REGION Network 6: #Do06 spare2
   RUNG wire#powerrail
      #Do06(Cmd :=, SimulationOn :=, MotorFeedbackInputSelection :=, MotorFeedbackInput :=, WaterSensorSelection :=, WaterSensorInput :=, AlwaysTrue := "AlwaysTRUE", AlwaysFalse := "AlwaysFALSE", OpenClose :=, Spare_3 :=, ValveFeedbackInputSelection :=, ValveFeedbackInput :=, Interlock := #Interlock, FBCheckDelay :=, WSCheckDelay :=, secs := "Sec_Pulse", AlarmAck :=, ModeSel :=, Fault :=, Reset :=, spare :=, spare_1 :=, spare_2 :=, OpFbTrip :=, OpWaterSensorTrip :=, FBCheckActualTime :=, WSCheckActualTime :=, Output =>, FeedBackTripAlarm =>, NoWaterFlowAlarm =>, LineColour =>, ValveColour =>, Mode =>, Status =>)
   END_RUNG
   // the same network as SCL:
   #Do06(AlwaysTrue := "AlwaysTRUE", AlwaysFalse := "AlwaysFALSE", Interlock := #Interlock, secs := "Sec_Pulse");   // "DigitalOutput"
END_REGION

REGION Network 7: #Do07spare3
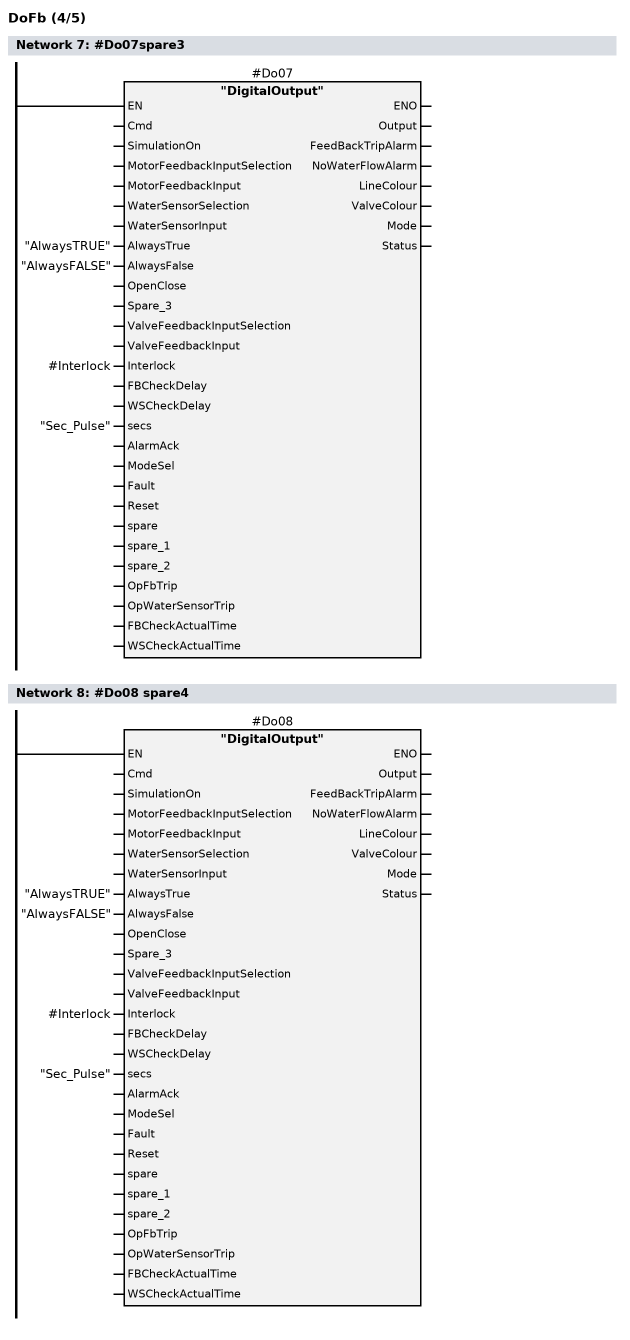
   RUNG wire#powerrail
      #Do07(Cmd :=, SimulationOn :=, MotorFeedbackInputSelection :=, MotorFeedbackInput :=, WaterSensorSelection :=, WaterSensorInput :=, AlwaysTrue := "AlwaysTRUE", AlwaysFalse := "AlwaysFALSE", OpenClose :=, Spare_3 :=, ValveFeedbackInputSelection :=, ValveFeedbackInput :=, Interlock := #Interlock, FBCheckDelay :=, WSCheckDelay :=, secs := "Sec_Pulse", AlarmAck :=, ModeSel :=, Fault :=, Reset :=, spare :=, spare_1 :=, spare_2 :=, OpFbTrip :=, OpWaterSensorTrip :=, FBCheckActualTime :=, WSCheckActualTime :=, Output =>, FeedBackTripAlarm =>, NoWaterFlowAlarm =>, LineColour =>, ValveColour =>, Mode =>, Status =>)
   END_RUNG
   // the same network as SCL:
   #Do07(AlwaysTrue := "AlwaysTRUE", AlwaysFalse := "AlwaysFALSE", Interlock := #Interlock, secs := "Sec_Pulse");   // "DigitalOutput"
END_REGION

REGION Network 8: #Do08 spare4
   RUNG wire#powerrail
      #Do08(Cmd :=, SimulationOn :=, MotorFeedbackInputSelection :=, MotorFeedbackInput :=, WaterSensorSelection :=, WaterSensorInput :=, AlwaysTrue := "AlwaysTRUE", AlwaysFalse := "AlwaysFALSE", OpenClose :=, Spare_3 :=, ValveFeedbackInputSelection :=, ValveFeedbackInput :=, Interlock := #Interlock, FBCheckDelay :=, WSCheckDelay :=, secs := "Sec_Pulse", AlarmAck :=, ModeSel :=, Fault :=, Reset :=, spare :=, spare_1 :=, spare_2 :=, OpFbTrip :=, OpWaterSensorTrip :=, FBCheckActualTime :=, WSCheckActualTime :=, Output =>, FeedBackTripAlarm =>, NoWaterFlowAlarm =>, LineColour =>, ValveColour =>, Mode =>, Status =>)
   END_RUNG
   // the same network as SCL:
   #Do08(AlwaysTrue := "AlwaysTRUE", AlwaysFalse := "AlwaysFALSE", Interlock := #Interlock, secs := "Sec_Pulse");   // "DigitalOutput"
END_REGION

REGION Network 9: ##Do09 spare5
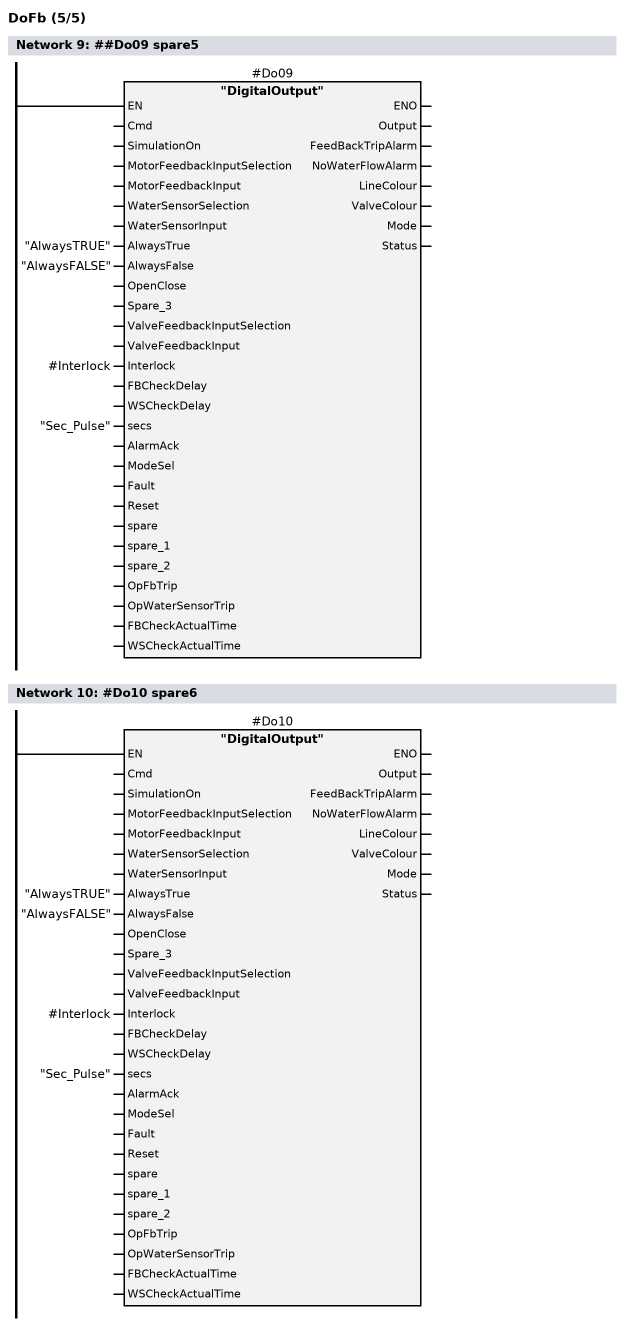
   RUNG wire#powerrail
      #Do09(Cmd :=, SimulationOn :=, MotorFeedbackInputSelection :=, MotorFeedbackInput :=, WaterSensorSelection :=, WaterSensorInput :=, AlwaysTrue := "AlwaysTRUE", AlwaysFalse := "AlwaysFALSE", OpenClose :=, Spare_3 :=, ValveFeedbackInputSelection :=, ValveFeedbackInput :=, Interlock := #Interlock, FBCheckDelay :=, WSCheckDelay :=, secs := "Sec_Pulse", AlarmAck :=, ModeSel :=, Fault :=, Reset :=, spare :=, spare_1 :=, spare_2 :=, OpFbTrip :=, OpWaterSensorTrip :=, FBCheckActualTime :=, WSCheckActualTime :=, Output =>, FeedBackTripAlarm =>, NoWaterFlowAlarm =>, LineColour =>, ValveColour =>, Mode =>, Status =>)
   END_RUNG
   // the same network as SCL:
   #Do09(AlwaysTrue := "AlwaysTRUE", AlwaysFalse := "AlwaysFALSE", Interlock := #Interlock, secs := "Sec_Pulse");   // "DigitalOutput"
END_REGION

REGION Network 10: #Do10 spare6
   RUNG wire#powerrail
      #Do10(Cmd :=, SimulationOn :=, MotorFeedbackInputSelection :=, MotorFeedbackInput :=, WaterSensorSelection :=, WaterSensorInput :=, AlwaysTrue := "AlwaysTRUE", AlwaysFalse := "AlwaysFALSE", OpenClose :=, Spare_3 :=, ValveFeedbackInputSelection :=, ValveFeedbackInput :=, Interlock := #Interlock, FBCheckDelay :=, WSCheckDelay :=, secs := "Sec_Pulse", AlarmAck :=, ModeSel :=, Fault :=, Reset :=, spare :=, spare_1 :=, spare_2 :=, OpFbTrip :=, OpWaterSensorTrip :=, FBCheckActualTime :=, WSCheckActualTime :=, Output =>, FeedBackTripAlarm =>, NoWaterFlowAlarm =>, LineColour =>, ValveColour =>, Mode =>, Status =>)
   END_RUNG
   // the same network as SCL:
   #Do10(AlwaysTrue := "AlwaysTRUE", AlwaysFalse := "AlwaysFALSE", Interlock := #Interlock, secs := "Sec_Pulse");   // "DigitalOutput"
END_REGION
END_FUNCTION_BLOCK

FUNCTION_BLOCK "DigitalOutput"   // FB4, LAD
TITLE = FB4
{ S7_Optimized_Access := 'FALSE' }
// DIGITAL OUTPUT
// stored: AutoNumber false, SetENOAutomatically false
   VAR_INPUT
      Cmd { ExternalVisible := 'False'} : Bool;
      SimulationOn { ExternalVisible := 'False'} : Bool;
      MotorFeedbackInputSelection { ExternalVisible := 'False'} : Bool;
      MotorFeedbackInput { ExternalVisible := 'False'} : Bool;
      WaterSensorSelection { ExternalVisible := 'False'} : Bool;
      WaterSensorInput { ExternalVisible := 'False'} : Bool;
      AlwaysTrue : Bool;
      AlwaysFalse : Bool;
      OpenClose : Bool;   // For Valve Only
      Spare_3 : Bool;   // For Valve Only
      ValveFeedbackInputSelection { ExternalVisible := 'False'} : Bool;
      ValveFeedbackInput { ExternalVisible := 'False'} : Bool;
      Interlock : Bool;
      FBCheckDelay { ExternalVisible := 'False'} : Int;
      WSCheckDelay { ExternalVisible := 'False'} : Int;
      secs { ExternalVisible := 'False'} : Bool;
      AlarmAck { ExternalVisible := 'False'} : Bool;
      ModeSel : Bool;   // 1=Man/ 0=Auto
      Fault : Bool;
      Reset : Bool;
      spare : Bool;
      spare_1 : Bool;
      spare_2 : Bool;
   END_VAR
   VAR_OUTPUT
      Output { ExternalVisible := 'False'} : Bool;
      FeedBackTripAlarm : Bool;
      NoWaterFlowAlarm : Bool;
      LineColour : DInt;
      ValveColour : DInt;
      Mode : DInt;   // Auto=0 , Manual=1
      Status : DInt;
   END_VAR
   VAR_IN_OUT
      OpFbTrip { ExternalVisible := 'False'} : Bool;
      OpWaterSensorTrip { ExternalVisible := 'False'} : Bool;
      FBCheckActualTime { ExternalVisible := 'False'} : Int;
      WSCheckActualTime { ExternalVisible := 'False'} : Int;
   END_VAR
   VAR
      ResetBtn { S7_SetPoint := 'True'} : TON_TIME;
   END_VAR
   VAR_TEMP   // added for the SCL form of the ladder/FBD networks
      _w1 : Bool;
      _w2 : Bool;
   END_VAR
BEGIN

REGION Network 1: #Output
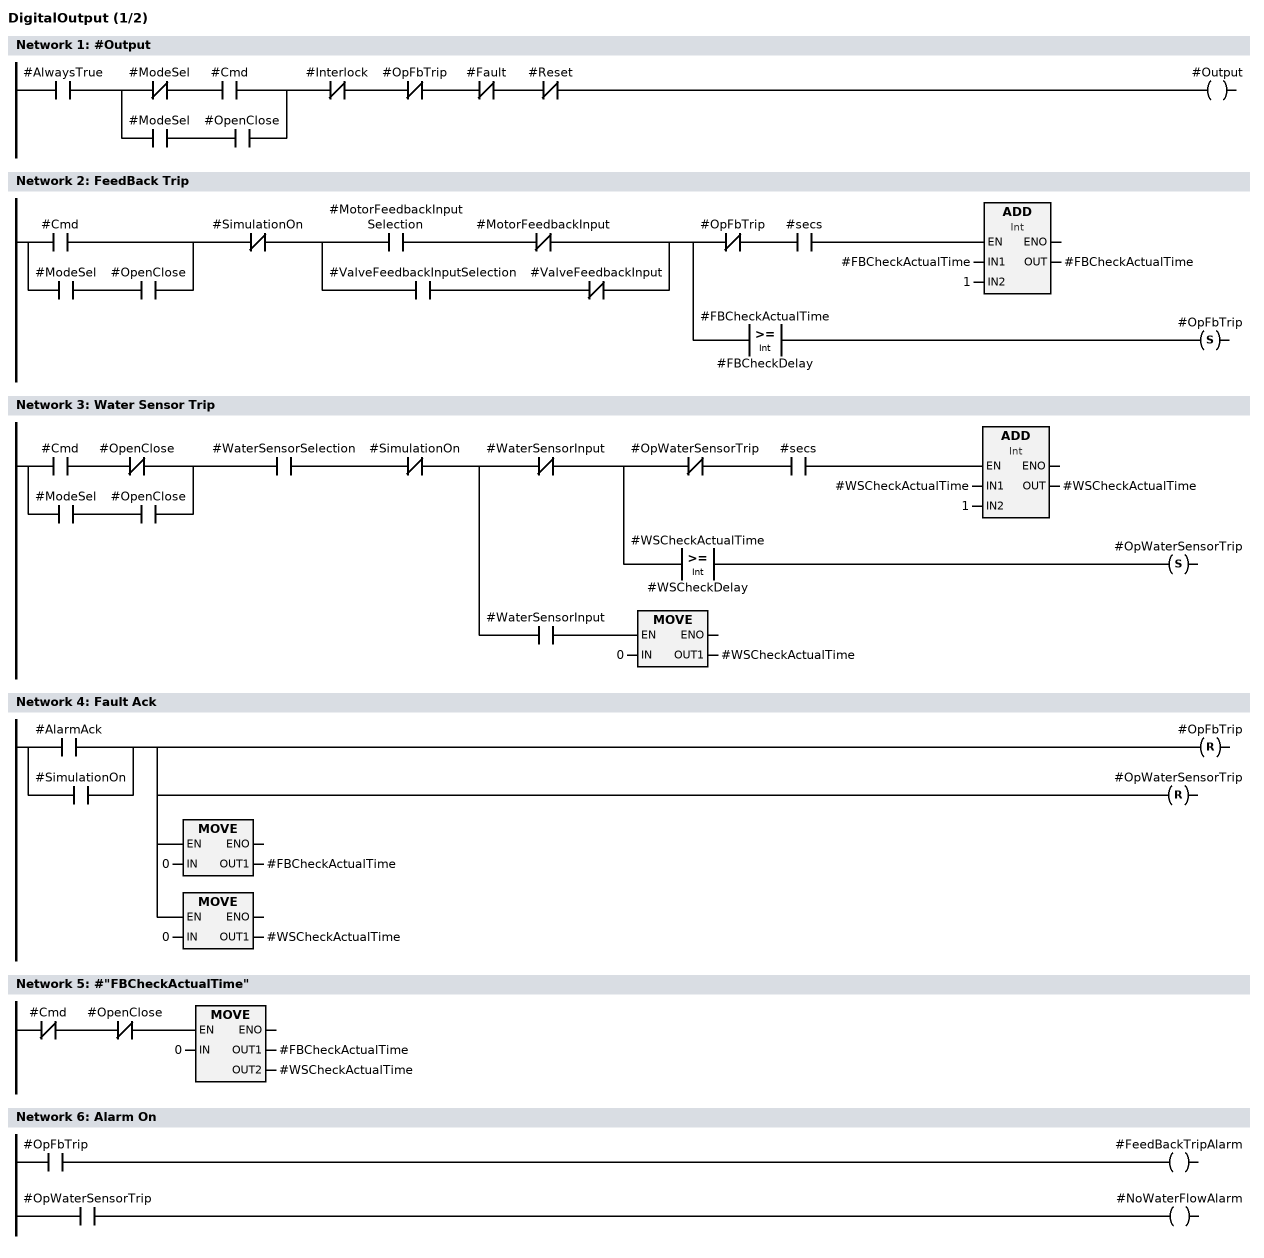
   RUNG wire#powerrail
      Contact( #AlwaysTrue )
      wire#w1
      I_Contact( #ModeSel )
      Contact( #Cmd )
      wire#w2
      I_Contact( #Interlock )
      I_Contact( #OpFbTrip )
      I_Contact( #Fault )
      I_Contact( #Reset )
      Coil( #Output )
   END_RUNG
   RUNG wire#w1
      Contact( #ModeSel )
      Contact( #OpenClose )
   END_RUNG wire#w2
   // the same network as SCL:
   #Output := #AlwaysTrue AND ((NOT #ModeSel AND #Cmd) OR (#ModeSel AND #OpenClose)) AND NOT #Interlock AND NOT #OpFbTrip AND NOT #Fault AND NOT #Reset;
END_REGION

REGION Network 2: FeedBack Trip
   RUNG wire#powerrail
      Contact( #Cmd )
      wire#w1
      I_Contact( #SimulationOn )
      wire#w2
      Contact( #MotorFeedbackInputSelection )
      I_Contact( #MotorFeedbackInput )
      wire#w3
      I_Contact( #OpFbTrip )
      Contact( #secs )
      { S7_Templates := "SrcType := Int"; S7_GenerateENO := "TRUE" } Add(in1 := #FBCheckActualTime, in2 := 1, out => #FBCheckActualTime)
   END_RUNG
   RUNG wire#powerrail
      Contact( #ModeSel )
      Contact( #OpenClose )
   END_RUNG wire#w1
   RUNG wire#w2
      Contact( #ValveFeedbackInputSelection )
      I_Contact( #ValveFeedbackInput )
   END_RUNG wire#w3
   RUNG wire#w3
      { S7_Templates := "SrcType := Int" } GE_Contact(in1 := #FBCheckActualTime, in2 := #FBCheckDelay)
      S_Coil( #OpFbTrip )
   END_RUNG
   // the same network as SCL:
   #_w1 := (#Cmd OR (#ModeSel AND #OpenClose)) AND NOT #SimulationOn AND ((#MotorFeedbackInputSelection AND NOT #MotorFeedbackInput) OR (#ValveFeedbackInputSelection AND NOT #ValveFeedbackInput));
   IF #_w1 AND NOT #OpFbTrip AND #secs THEN #FBCheckActualTime := #FBCheckActualTime + 1; END_IF;
   IF #_w1 AND (#FBCheckActualTime >= #FBCheckDelay) THEN #OpFbTrip := TRUE; END_IF;
END_REGION

REGION Network 3: Water Sensor Trip
   RUNG wire#powerrail
      Contact( #Cmd )
      I_Contact( #OpenClose )
      wire#w1
      Contact( #WaterSensorSelection )
      I_Contact( #SimulationOn )
      wire#w2
      I_Contact( #WaterSensorInput )
      wire#w3
      I_Contact( #OpWaterSensorTrip )
      Contact( #secs )
      { S7_Templates := "SrcType := Int"; S7_GenerateENO := "TRUE" } Add(in1 := #WSCheckActualTime, in2 := 1, out => #WSCheckActualTime)
   END_RUNG
   RUNG wire#powerrail
      Contact( #ModeSel )
      Contact( #OpenClose )
   END_RUNG wire#w1
   RUNG wire#w3
      { S7_Templates := "SrcType := Int" } GE_Contact(in1 := #WSCheckActualTime, in2 := #WSCheckDelay)
      S_Coil( #OpWaterSensorTrip )
   END_RUNG
   RUNG wire#w2
      Contact( #WaterSensorInput )
      { S7_GenerateENO := "TRUE" } Move(in := 0, out1 => #WSCheckActualTime)
   END_RUNG
   // the same network as SCL:
   #_w1 := ((#Cmd AND NOT #OpenClose) OR (#ModeSel AND #OpenClose)) AND #WaterSensorSelection AND NOT #SimulationOn;
   #_w2 := #_w1 AND NOT #WaterSensorInput;
   IF #_w2 AND NOT #OpWaterSensorTrip AND #secs THEN #WSCheckActualTime := #WSCheckActualTime + 1; END_IF;
   IF #_w2 AND (#WSCheckActualTime >= #WSCheckDelay) THEN #OpWaterSensorTrip := TRUE; END_IF;
   IF #_w1 AND #WaterSensorInput THEN #WSCheckActualTime := 0; END_IF;
END_REGION

REGION Network 4: Fault Ack
   RUNG wire#powerrail
      Contact( #AlarmAck )
      wire#w1
      R_Coil( #OpFbTrip )
   END_RUNG
   RUNG wire#powerrail
      Contact( #SimulationOn )
   END_RUNG wire#w1
   RUNG wire#w1
      R_Coil( #OpWaterSensorTrip )
   END_RUNG
   RUNG wire#w1
      { S7_GenerateENO := "TRUE" } Move(in := 0, out1 => #FBCheckActualTime)
   END_RUNG
   RUNG wire#w1
      { S7_GenerateENO := "TRUE" } Move(in := 0, out1 => #WSCheckActualTime)
   END_RUNG
   // the same network as SCL:
   IF #AlarmAck OR #SimulationOn THEN
       #OpFbTrip := FALSE;
       #OpWaterSensorTrip := FALSE;
       #FBCheckActualTime := 0;
       #WSCheckActualTime := 0;
   END_IF;
END_REGION

REGION Network 5: #"FBCheckActualTime"
   RUNG wire#powerrail
      I_Contact( #Cmd )
      I_Contact( #OpenClose )
      { S7_GenerateENO := "TRUE" } Move(in := 0, out1 => #FBCheckActualTime, out2 => #WSCheckActualTime)
   END_RUNG
   // the same network as SCL:
   IF NOT #Cmd AND NOT #OpenClose THEN
       #FBCheckActualTime := 0;
       #WSCheckActualTime := 0;
   END_IF;
END_REGION

REGION Network 6: Alarm On
   RUNG wire#powerrail
      Contact( #OpFbTrip )
      Coil( #FeedBackTripAlarm )
   END_RUNG
   RUNG wire#powerrail
      Contact( #OpWaterSensorTrip )
      Coil( #NoWaterFlowAlarm )
   END_RUNG
   // the same network as SCL:
   #FeedBackTripAlarm := #OpFbTrip;
   #NoWaterFlowAlarm := #OpWaterSensorTrip;
END_REGION

REGION Network 7: Valve Colour
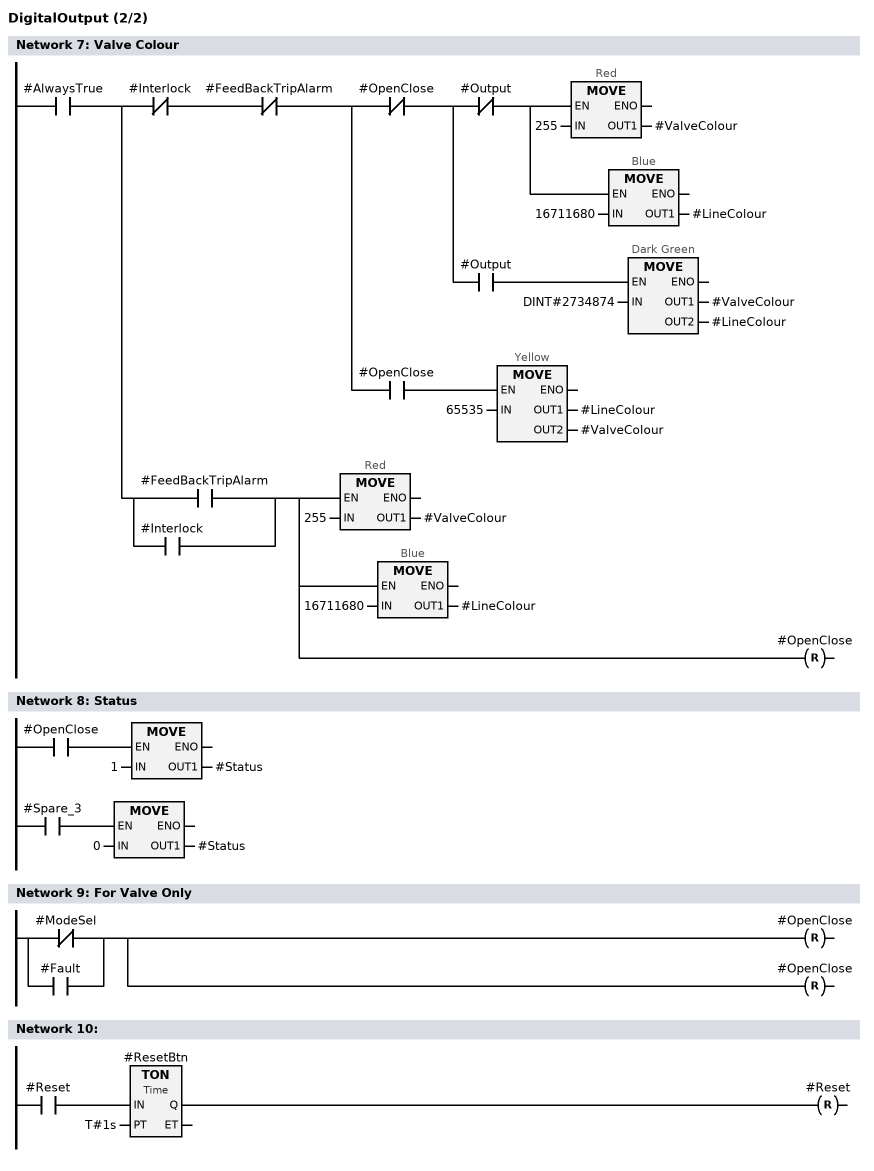
   RUNG wire#powerrail
      Contact( #AlwaysTrue )
      wire#w1
      I_Contact( #Interlock )
      I_Contact( #FeedBackTripAlarm )
      wire#w2
      I_Contact( #OpenClose )
      wire#w3
      I_Contact( #Output )
      wire#w4
      Move(in := 255, out1 => #ValveColour)   // Red
   END_RUNG
   RUNG wire#w4
      Move(in := 16711680, out1 => #LineColour)   // Blue
   END_RUNG
   RUNG wire#w3
      Contact( #Output )
      Move(in := DINT#2734874, out1 => #ValveColour, out2 => #LineColour)   // Dark Green
   END_RUNG
   RUNG wire#w2
      Contact( #OpenClose )
      Move(in := 65535, out1 => #LineColour, out2 => #ValveColour)   // Yellow
   END_RUNG
   RUNG wire#w1
      Contact( #FeedBackTripAlarm )
      wire#w5
      Move(in := 255, out1 => #ValveColour)   // Red
   END_RUNG
   RUNG wire#w1
      Contact( #Interlock )
   END_RUNG wire#w5
   RUNG wire#w5
      Move(in := 16711680, out1 => #LineColour)   // Blue
   END_RUNG
   RUNG wire#w5
      R_Coil( #OpenClose )
   END_RUNG
   // the same network as SCL:
   #_w1 := #AlwaysTrue AND NOT #Interlock AND NOT #FeedBackTripAlarm;
   #_w2 := #_w1 AND NOT #OpenClose;
   IF #_w2 AND NOT #Output THEN
       #ValveColour := 255;   // Red
       #LineColour := 16711680;   // Blue
   END_IF;
   IF #_w2 AND #Output THEN
       #ValveColour := DINT#2734874;   // Dark Green
       #LineColour := DINT#2734874;
   END_IF;
   IF #_w1 AND #OpenClose THEN
       #LineColour := 65535;   // Yellow
       #ValveColour := 65535;
   END_IF;
   IF #AlwaysTrue AND (#FeedBackTripAlarm OR #Interlock) THEN
       #ValveColour := 255;   // Red
       #LineColour := 16711680;   // Blue
       #OpenClose := FALSE;
   END_IF;
END_REGION

REGION Network 8: Status
   RUNG wire#powerrail
      Contact( #OpenClose )
      Move(in := 1, out1 => #Status)
   END_RUNG
   RUNG wire#powerrail
      Contact( #Spare_3 )
      Move(in := 0, out1 => #Status)
   END_RUNG
   // the same network as SCL:
   IF #OpenClose THEN #Status := 1; END_IF;
   IF #Spare_3 THEN #Status := 0; END_IF;
END_REGION

REGION Network 9: For Valve Only
   RUNG wire#powerrail
      I_Contact( #ModeSel )
      wire#w1
      R_Coil( #OpenClose )
   END_RUNG
   RUNG wire#powerrail
      Contact( #Fault )
   END_RUNG wire#w1
   RUNG wire#w1
      R_Coil( #OpenClose )
   END_RUNG
   // the same network as SCL:
   IF NOT #ModeSel OR #Fault THEN
       #OpenClose := FALSE;
       #OpenClose := FALSE;
   END_IF;
END_REGION

REGION Network 10
   RUNG wire#powerrail
      Contact( #Reset )
      { S7_Templates := "time_type := Time" } #ResetBtn.TON(pt := T#1s, et =>)
      R_Coil( #Reset )
   END_RUNG
   // the same network as SCL:
   #ResetBtn(IN := #Reset, PT := T#1s);   // TON
   IF #ResetBtn.Q THEN #Reset := FALSE; END_IF;
END_REGION
END_FUNCTION_BLOCK

FUNCTION_BLOCK "TIMER"   // FB6, LAD
{ S7_Optimized_Access := 'FALSE' }
// stored: SetENOAutomatically false
   VAR_INPUT
      TIME_START : Bool;
      TIME_PULSE : Bool;
      TIME_TRSET : Bool;
      MINI_ENABLE : Bool;
      TIME_IN_MINI : DInt;
      TIME_IN_SEC : DInt;
   END_VAR
   VAR_OUTPUT
      DONE_BIT : Bool;
      ES_MINIT : DInt;
      ES_SEC : DInt;
   END_VAR
   VAR_IN_OUT
      TEMP_1 : DInt;
      TEMP_5 : DInt;
      TEMP_2 : DInt;
      TEMP_3 : DInt;
      TEMP_BIT_1 : Bool;
      TEMP_BIT_2 : Bool;
   END_VAR
   VAR_TEMP   // added for the SCL form of the ladder/FBD networks
      _w1 : Bool;
   END_VAR
BEGIN

REGION Network 1
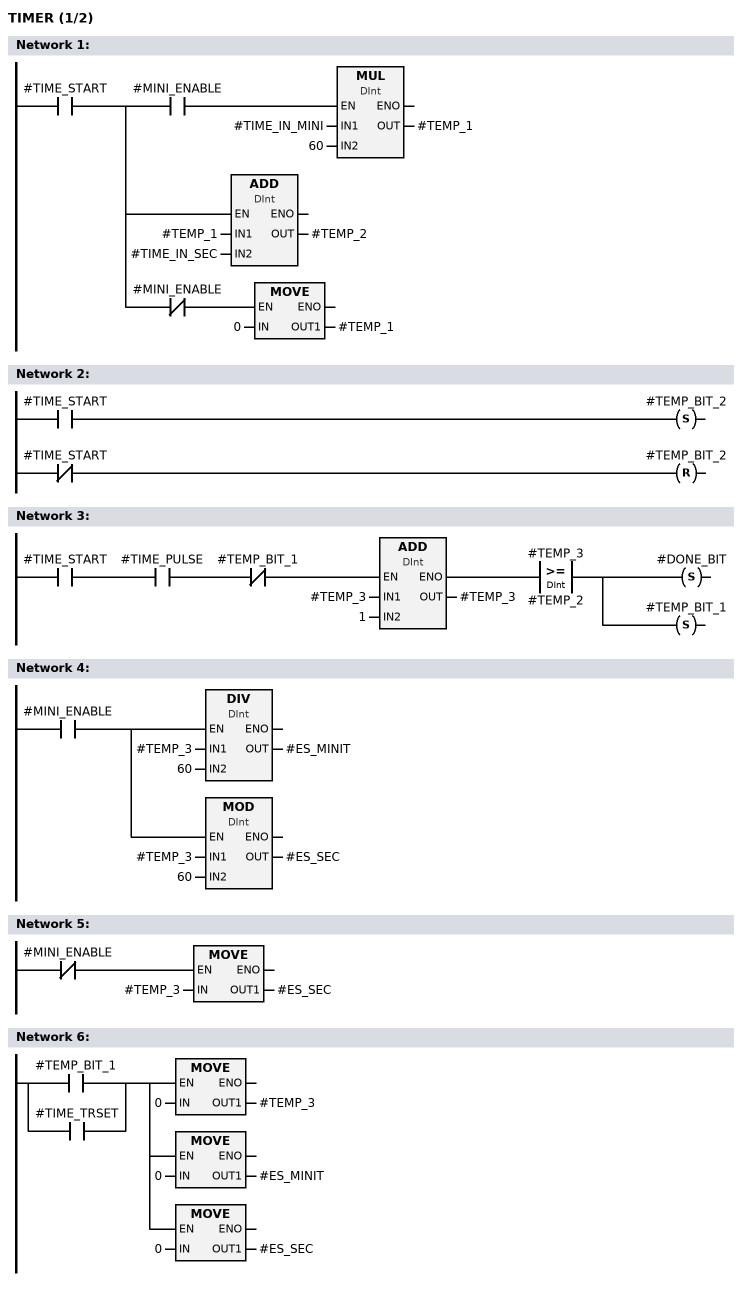
   RUNG wire#powerrail
      Contact( #TIME_START )
      wire#w1
      Contact( #MINI_ENABLE )
      { S7_Templates := "SrcType := DInt"; S7_GenerateENO := "TRUE" } Mul(in1 := #TIME_IN_MINI, in2 := 60, out => #TEMP_1)
   END_RUNG
   RUNG wire#w1
      { S7_Templates := "SrcType := DInt"; S7_GenerateENO := "TRUE" } Add(in1 := #TEMP_1, in2 := #TIME_IN_SEC, out => #TEMP_2)
   END_RUNG
   RUNG wire#w1
      I_Contact( #MINI_ENABLE )
      { S7_GenerateENO := "TRUE" } Move(in := 0, out1 => #TEMP_1)
   END_RUNG
   // the same network as SCL:
   IF #TIME_START AND #MINI_ENABLE THEN #TEMP_1 := #TIME_IN_MINI * 60; END_IF;
   IF #TIME_START THEN #TEMP_2 := #TEMP_1 + #TIME_IN_SEC; END_IF;
   IF #TIME_START AND NOT #MINI_ENABLE THEN #TEMP_1 := 0; END_IF;
END_REGION

REGION Network 2
   RUNG wire#powerrail
      Contact( #TIME_START )
      S_Coil( #TEMP_BIT_2 )
   END_RUNG
   RUNG wire#powerrail
      I_Contact( #TIME_START )
      R_Coil( #TEMP_BIT_2 )
   END_RUNG
   // the same network as SCL:
   IF #TIME_START THEN #TEMP_BIT_2 := TRUE; END_IF;
   IF NOT #TIME_START THEN #TEMP_BIT_2 := FALSE; END_IF;
END_REGION

REGION Network 3
   RUNG wire#powerrail
      Contact( #TIME_START )
      Contact( #TIME_PULSE )
      I_Contact( #TEMP_BIT_1 )
      { S7_Templates := "SrcType := DInt"; S7_GenerateENO := "TRUE" } Add(in1 := #TEMP_3, in2 := 1, out => #TEMP_3)
      { S7_Templates := "SrcType := DInt" } GE_Contact(in1 := #TEMP_3, in2 := #TEMP_2)
      wire#w1
      S_Coil( #DONE_BIT )
   END_RUNG
   RUNG wire#w1
      S_Coil( #TEMP_BIT_1 )
   END_RUNG
   // the same network as SCL:
   // ENO of a box is taken as its EN; it also drops when the box reports an error
   #_w1 := #TIME_START AND #TIME_PULSE AND NOT #TEMP_BIT_1;
   IF #_w1 THEN #TEMP_3 := #TEMP_3 + 1; END_IF;
   IF #_w1 AND (#TEMP_3 >= #TEMP_2) THEN
       #DONE_BIT := TRUE;
       #TEMP_BIT_1 := TRUE;
   END_IF;
END_REGION

REGION Network 4
   RUNG wire#powerrail
      Contact( #MINI_ENABLE )
      wire#w1
      { S7_Templates := "SrcType := DInt"; S7_GenerateENO := "TRUE" } Div(in1 := #TEMP_3, in2 := 60, out => #ES_MINIT)
   END_RUNG
   RUNG wire#w1
      { S7_Templates := "SrcType := DInt"; S7_GenerateENO := "TRUE" } Mod(in1 := #TEMP_3, in2 := 60, out => #ES_SEC)
   END_RUNG
   // the same network as SCL:
   IF #MINI_ENABLE THEN
       #ES_MINIT := #TEMP_3 / 60;
       #ES_SEC := #TEMP_3 MOD 60;
   END_IF;
END_REGION

REGION Network 5
   RUNG wire#powerrail
      I_Contact( #MINI_ENABLE )
      { S7_GenerateENO := "TRUE" } Move(in := #TEMP_3, out1 => #ES_SEC)
   END_RUNG
   // the same network as SCL:
   IF NOT #MINI_ENABLE THEN #ES_SEC := #TEMP_3; END_IF;
END_REGION

REGION Network 6
   RUNG wire#powerrail
      Contact( #TEMP_BIT_1 )
      wire#w1
      { S7_GenerateENO := "TRUE" } Move(in := 0, out1 => #TEMP_3)
   END_RUNG
   RUNG wire#powerrail
      Contact( #TIME_TRSET )
   END_RUNG wire#w1
   RUNG wire#w1
      { S7_GenerateENO := "TRUE" } Move(in := 0, out1 => #ES_MINIT)
   END_RUNG
   RUNG wire#w1
      { S7_GenerateENO := "TRUE" } Move(in := 0, out1 => #ES_SEC)
   END_RUNG
   // the same network as SCL:
   IF #TEMP_BIT_1 OR #TIME_TRSET THEN
       #TEMP_3 := 0;
       #ES_MINIT := 0;
       #ES_SEC := 0;
   END_IF;
END_REGION

REGION Network 7
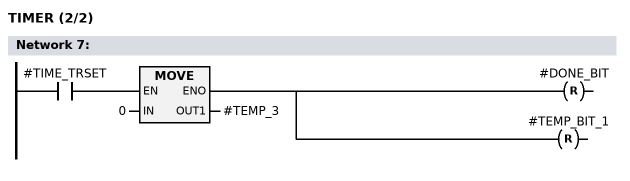
   RUNG wire#powerrail
      Contact( #TIME_TRSET )
      { S7_GenerateENO := "TRUE" } Move(in := 0, out1 => #TEMP_3)
      wire#w1
      R_Coil( #DONE_BIT )
   END_RUNG
   RUNG wire#w1
      R_Coil( #TEMP_BIT_1 )
   END_RUNG
   // the same network as SCL:
   // ENO of a box is taken as its EN; it also drops when the box reports an error
   IF #TIME_TRSET THEN
       #TEMP_3 := 0;
       #DONE_BIT := FALSE;
       #TEMP_BIT_1 := FALSE;
   END_IF;
END_REGION
END_FUNCTION_BLOCK

FUNCTION "FaceplateFc" : Void   // FC102, LAD
{ S7_Optimized_Access := 'TRUE' }
// stored: AutoNumber false, SetENOAutomatically false
BEGIN

REGION Network 1 (SCL): Valve Open
   "ValveManualMode".Cv01 := "DO_FaceplateDb".Cv01.ValveOpen;
   "ValveManualMode".Cv01 := "DO_FaceplateDb".Cv01.ValveOpen;
   "ValveManualMode".Cv02 := "DO_FaceplateDb".Cv02.ValveOpen;
   "ValveManualMode".Cv03 := "DO_FaceplateDb".Cv03.ValveOpen;
   "ValveManualMode".Cv04 := "DO_FaceplateDb".Cv04.ValveOpen;
   "ValveManualMode".Cv05 := "DO_FaceplateDb".Cv05.ValveOpen;
   "ValveManualMode".Cv06 := "DO_FaceplateDb".Cv06.ValveOpen;
   "ValveManualMode".Cv07 := "DO_FaceplateDb".Cv07.ValveOpen;
   "ValveManualMode".Cv08 := "DO_FaceplateDb".Cv08.ValveOpen;
   "ValveManualMode".Cv09 := "DO_FaceplateDb".Cv09.ValveOpen;
   "ValveManualMode".Cv10 := "DO_FaceplateDb".Cv10.ValveOpen;
   "ValveManualMode".Cv11 := "DO_FaceplateDb".Cv11.ValveOpen;
   "ValveManualMode".Cv12 := "DO_FaceplateDb".Cv12.ValveOpen;
   "ValveManualMode".Cv13 := "DO_FaceplateDb".Cv13.ValveOpen;
   "ValveManualMode".Cv14 := "DO_FaceplateDb".Cv14.ValveOpen;
   "ValveManualMode".Cv15 := "DO_FaceplateDb".Cv15.ValveOpen;
   "ValveManualMode".Cv16 := "DO_FaceplateDb".Cv16.ValveOpen;
   "ValveManualMode".Cv17 := "DO_FaceplateDb".Cv17.ValveOpen;
   "ValveManualMode".Cv18 := "DO_FaceplateDb".Cv18.ValveOpen;
   "ValveManualMode".Cv19 := "DO_FaceplateDb".Cv19.ValveOpen;
   "ValveManualMode".Cv20 := "DO_FaceplateDb".Cv20.ValveOpen;
   "ValveManualMode".Cv21 := "DO_FaceplateDb".Cv21.ValveOpen;
   "ValveManualMode".Cv22 := "DO_FaceplateDb".Cv22.ValveOpen;
   "ValveManualMode".Cv23 := "DO_FaceplateDb".Cv23.ValveOpen;
   "ValveManualMode".Cv24 := "DO_FaceplateDb".Cv24.ValveOpen;
   "ValveManualMode".Cv25 := "DO_FaceplateDb".Cv25.ValveOpen;
   "ValveManualMode".Cv26 := "DO_FaceplateDb".Cv26.ValveOpen;
   "ValveManualMode".Cv27 := "DO_FaceplateDb".Cv27.ValveOpen;
   "ValveManualMode".Cv28 := "DO_FaceplateDb".Cv28.ValveOpen;
   "ValveManualMode".Cv29 := "DO_FaceplateDb".Cv29.ValveOpen;
   "ValveManualMode".Cv30 := "DO_FaceplateDb".Cv30.ValveOpen;
   "ValveManualMode".Cv31 := "DO_FaceplateDb".Cv31.ValveOpen;
   "ValveManualMode".Cv32 := "DO_FaceplateDb".Cv32.ValveOpen;
   "ValveManualMode".Cv33 := "DO_FaceplateDb".Cv33.ValveOpen;
   "ValveManualMode".Cv34 := "DO_FaceplateDb".Cv34.ValveOpen;
   "ValveManualMode".Cv35 := "DO_FaceplateDb".Cv35.ValveOpen;
   "ValveManualMode".Cv36 := "DO_FaceplateDb".Cv36.ValveOpen;
   "ValveManualMode".Cv37 := "DO_FaceplateDb".Cv37.ValveOpen;
   "ValveManualMode".Cv38 := "DO_FaceplateDb".Cv38.ValveOpen;
   "ValveManualMode".Cv39 := "DO_FaceplateDb".Cv39.ValveOpen;
   "ValveManualMode".Cv40 := "DO_FaceplateDb".Cv40.ValveOpen;
   "ValveManualMode".Cv41 := "DO_FaceplateDb".Cv41.ValveOpen;
   "ValveManualMode".Cv42 := "DO_FaceplateDb".Cv42.ValveOpen;
   "ValveManualMode".Cv43 := "DO_FaceplateDb".Cv43.ValveOpen;
   "ValveManualMode".Cv44 := "DO_FaceplateDb".Cv44.ValveOpen;
   "ValveManualMode".Cv45 := "DO_FaceplateDb".Cv45.ValveOpen;
   "ValveManualMode".Cv46 := "DO_FaceplateDb".Cv46.ValveOpen;
   "ValveManualMode".Cv47 := "DO_FaceplateDb".Cv47.ValveOpen;
   "ValveManualMode".Cv48 := "DO_FaceplateDb".Cv48.ValveOpen;
   "ValveManualMode".Cv49 := "DO_FaceplateDb".Cv49.ValveOpen;
   "ValveManualMode".Cv50 := "DO_FaceplateDb".Cv50.ValveOpen;
   "ValveManualMode".Cv51 := "DO_FaceplateDb".Cv51.ValveOpen;
   "ValveManualMode".Cv52 := "DO_FaceplateDb".Cv52.ValveOpen;
   "ValveManualMode".Cv53 := "DO_FaceplateDb".Cv53.ValveOpen;
   "ValveManualMode".Cv54 := "DO_FaceplateDb".Cv54.ValveOpen;
   "ValveManualMode".Cv55 := "DO_FaceplateDb".Cv55.ValveOpen;
   "ValveManualMode".Cv56 := "DO_FaceplateDb".Cv56.ValveOpen;
   "ValveManualMode".Cv57 := "DO_FaceplateDb".Cv57.ValveOpen;
   "ValveManualMode".Cv58 := "DO_FaceplateDb".Cv58.ValveOpen;
   "ValveManualMode".Cv59 := "DO_FaceplateDb".Cv59.ValveOpen;
   "ValveManualMode".Cv60 := "DO_FaceplateDb".Cv60.ValveOpen;
   "ValveManualMode".Cv61 := "DO_FaceplateDb".Cv61.ValveOpen;
   "ValveManualMode".Cv62 := "DO_FaceplateDb".Cv62.ValveOpen;
   "ValveManualMode".Cv63 := "DO_FaceplateDb".Cv63.ValveOpen;
   "ValveManualMode".Cv64 := "DO_FaceplateDb".Cv64.ValveOpen;
   "ValveManualMode".Fbov01 := "DO_FaceplateDb".Fbov01.ValveOpen;
END_REGION

REGION Network 2 (SCL): Pump Command
   "DoManualModeDb".Mm01Cmd :="DO_FaceplateDb"."Mm01 Ref".ValveOpen;
   "DoManualModeDb".Cp01Cmd := "DO_FaceplateDb"."Cp01 Ref".ValveOpen;


   //"DoDb".Do01.OpenClose := "DO_FaceplateDb"."Mm01 Ref".ValveOpen;
   //"DoDb".Do02.OpenClose := "DO_FaceplateDb"."Cp01 Ref".ValveOpen;
END_REGION

REGION Network 3 (SCL): Analog Output
   //Actual Rpm

   "Ao_Faceplate_Db".Mm01Ref.ActualRpm := "AoDb".Ao01.ActualRpm;
   "Ao_Faceplate_Db".Cp01Ref.ActualRpm:= "AoDb".Ao02.ActualRpm;


   //Min. Opeating Rpm
   // "AoDb".Ao01.MinOperatingRpm := "Ao_Faceplate_Db".CP01.MinOperating;
   //"AoDb".Ao02.MinOperatingRpm := "Ao_Faceplate_Db".MM01.MinOperating;
   "Ao_Faceplate_Db".Mm01Ref.MinOperating:= "AoDb".Ao01.MinOperatingRpm;
   "Ao_Faceplate_Db".Cp01Ref.MinOperating := "AoDb".Ao02.MinOperatingRpm;

   //Max. Operating Rpm
   "Ao_Faceplate_Db".Mm01Ref.MaxOperating:=  "AoDb".Ao01.MaxOperatingRpm;
   "Ao_Faceplate_Db".Cp01Ref.MaxOperating:= "AoDb".Ao02.MaxOperatingRpm;

   //Maximum Rpm
   // "AoDb".Ao01.MaxRpm := "Ao_Faceplate_Db".CP01.Maximum;
   // "AoDb".Ao02.MaxRpm := "Ao_Faceplate_Db".MM01.Maximum;
   "Ao_Faceplate_Db".Mm01Ref.Maximum:= "AoDb".Ao01.MaxRpm;
   "Ao_Faceplate_Db".Cp01Ref.Maximum:= "AoDb".Ao02.MaxRpm;

   //Manual Rpm
   // "AoDb".Ao01.ManualRpm := "Ao_Faceplate_Db".CP01.Manual;
   // "AoDb".Ao02.ManualRpm := "Ao_Faceplate_Db".MM01.Manual;
   "Ao_Faceplate_Db".Mm01Ref.Manual := "AoDb".Ao01.ManualRpm;
   "Ao_Faceplate_Db".Cp01Ref.Manual:= "AoDb".Ao02.ManualRpm;
END_REGION

REGION Network 4 (SCL): Analog Input
   // Moving Int value for units, 0 - Degree Celcius, 1 - bar, 2 - 

   // //"Ai_Faceplate_Db".Ai01.Unit := 0; spare
   // //"Ai_Faceplate_Db".Ai02.Unit := 0; spare
   // "Ai_Faceplate_Db".Ai03.Unit := 0;
   // "Ai_Faceplate_Db".Ai04.Unit := 0;
   // "Ai_Faceplate_Db".Ai05.Unit := 0;
   // "Ai_Faceplate_Db".Ai06.Unit := 0;
   // "Ai_Faceplate_Db".Ai07.Unit := 0;
   // "Ai_Faceplate_Db".Ai08.Unit := 1;
   // "Ai_Faceplate_Db".Ai09.Unit := 2;
   // "Ai_Faceplate_Db".Ai10.Unit := 3;
   // "Ai_Faceplate_Db".Ai11.Unit := 4;
END_REGION

REGION Network 5 (SCL)
   // "ValveDb".Cv01.OpenClose := "DO_FaceplateDb".Cv01.ValveOpen;
END_REGION
END_FUNCTION

FUNCTION "AlarmsFc" : Void   // FC181, LAD
{ S7_Optimized_Access := 'TRUE' }
// stored: AutoNumber false, SetENOAutomatically false
   VAR_TEMP   // added for the SCL form of the ladder/FBD networks
      _w1 : Bool;
      _w2 : Bool;
      _w3 : Bool;
      _w4 : Bool;
      _w5 : Bool;
      _w6 : Bool;
      _w7 : Bool;
      _w8 : Bool;
      _w9 : Bool;
      _w10 : Bool;
      _w11 : Bool;
      _w12 : Bool;
      _w13 : Bool;
      _w14 : Bool;
      _w15 : Bool;
      _w16 : Bool;
      _w17 : Bool;
      _w18 : Bool;
      _w19 : Bool;
      _w20 : Bool;
      _w21 : Bool;
      _w22 : Bool;
      _w23 : Bool;
      _w24 : Bool;
      _w25 : Bool;
      _w26 : Bool;
      _w27 : Bool;
      _w28 : Bool;
      _w29 : Bool;
      _w30 : Bool;
      _w31 : Bool;
      _w32 : Bool;
      _w33 : Bool;
      _w34 : Bool;
      _w35 : Bool;
      _w36 : Bool;
      _w37 : Bool;
      _w38 : Bool;
      _w39 : Bool;
      _w40 : Bool;
      _w41 : Bool;
      _w42 : Bool;
      _w43 : Bool;
      _w44 : Bool;
      _w45 : Bool;
      _w46 : Bool;
   END_VAR
BEGIN

REGION Network 1: "SafetyAlarms".ControlKeyOff
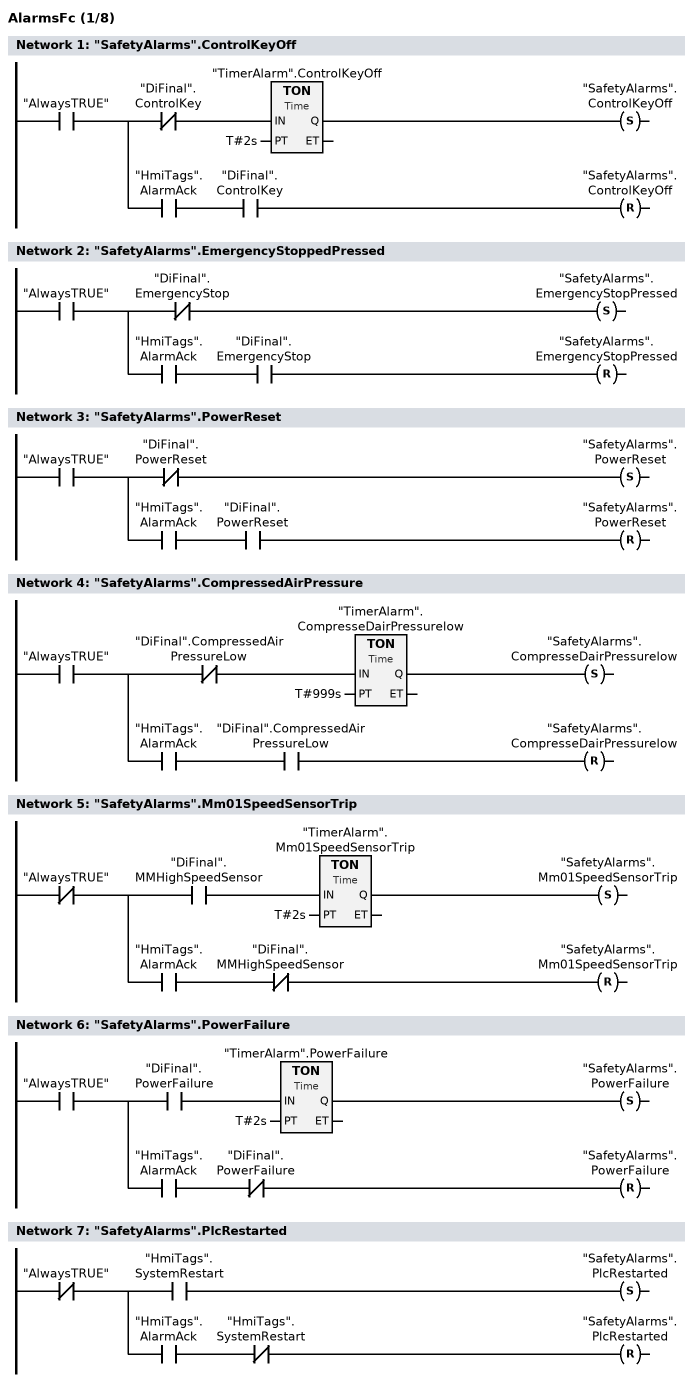
   RUNG wire#powerrail
      Contact( "AlwaysTRUE" )
      wire#w1
      I_Contact( "DiFinal".ControlKey )
      { S7_Templates := "time_type := Time" } "TimerAlarm".ControlKeyOff.TON(pt := T#2s, et =>)
      S_Coil( "SafetyAlarms".ControlKeyOff )
   END_RUNG
   RUNG wire#w1
      Contact( "HmiTags".AlarmAck )
      Contact( "DiFinal".ControlKey )
      R_Coil( "SafetyAlarms".ControlKeyOff )
   END_RUNG
   // the same network as SCL:
   "TimerAlarm".ControlKeyOff.TON(IN := "AlwaysTRUE" AND NOT "DiFinal".ControlKey, PT := T#2s);
   IF "TimerAlarm".ControlKeyOff.Q THEN "SafetyAlarms".ControlKeyOff := TRUE; END_IF;
   IF "AlwaysTRUE" AND "HmiTags".AlarmAck AND "DiFinal".ControlKey THEN
       "SafetyAlarms".ControlKeyOff := FALSE;
   END_IF;
END_REGION

REGION Network 2: "SafetyAlarms".EmergencyStoppedPressed
   RUNG wire#powerrail
      Contact( "AlwaysTRUE" )
      wire#w1
      I_Contact( "DiFinal".EmergencyStop )
      S_Coil( "SafetyAlarms".EmergencyStopPressed )
   END_RUNG
   RUNG wire#w1
      Contact( "HmiTags".AlarmAck )
      Contact( "DiFinal".EmergencyStop )
      R_Coil( "SafetyAlarms".EmergencyStopPressed )
   END_RUNG
   // the same network as SCL:
   IF "AlwaysTRUE" AND NOT "DiFinal".EmergencyStop THEN "SafetyAlarms".EmergencyStopPressed := TRUE; END_IF;
   IF "AlwaysTRUE" AND "HmiTags".AlarmAck AND "DiFinal".EmergencyStop THEN
       "SafetyAlarms".EmergencyStopPressed := FALSE;
   END_IF;
END_REGION

REGION Network 3: "SafetyAlarms".PowerReset
   RUNG wire#powerrail
      Contact( "AlwaysTRUE" )
      wire#w1
      I_Contact( "DiFinal".PowerReset )
      S_Coil( "SafetyAlarms".PowerReset )
   END_RUNG
   RUNG wire#w1
      Contact( "HmiTags".AlarmAck )
      Contact( "DiFinal".PowerReset )
      R_Coil( "SafetyAlarms".PowerReset )
   END_RUNG
   // the same network as SCL:
   IF "AlwaysTRUE" AND NOT "DiFinal".PowerReset THEN "SafetyAlarms".PowerReset := TRUE; END_IF;
   IF "AlwaysTRUE" AND "HmiTags".AlarmAck AND "DiFinal".PowerReset THEN
       "SafetyAlarms".PowerReset := FALSE;
   END_IF;
END_REGION

REGION Network 4: "SafetyAlarms".CompressedAirPressure
   RUNG wire#powerrail
      Contact( "AlwaysTRUE" )
      wire#w1
      I_Contact( "DiFinal".CompressedAirPressureLow )
      { S7_Templates := "time_type := Time" } "TimerAlarm".CompresseDairPressurelow.TON(pt := T#999s, et =>)
      S_Coil( "SafetyAlarms".CompresseDairPressurelow )
   END_RUNG
   RUNG wire#w1
      Contact( "HmiTags".AlarmAck )
      Contact( "DiFinal".CompressedAirPressureLow )
      R_Coil( "SafetyAlarms".CompresseDairPressurelow )
   END_RUNG
   // the same network as SCL:
   "TimerAlarm".CompresseDairPressurelow.TON(IN := "AlwaysTRUE" AND NOT "DiFinal".CompressedAirPressureLow,
                           PT := T#999s);
   IF "TimerAlarm".CompresseDairPressurelow.Q THEN "SafetyAlarms".CompresseDairPressurelow := TRUE; END_IF;
   IF "AlwaysTRUE" AND "HmiTags".AlarmAck AND "DiFinal".CompressedAirPressureLow THEN
       "SafetyAlarms".CompresseDairPressurelow := FALSE;
   END_IF;
END_REGION

REGION Network 5: "SafetyAlarms".Mm01SpeedSensorTrip
   RUNG wire#powerrail
      I_Contact( "AlwaysTRUE" )
      wire#w1
      Contact( "DiFinal".MMHighSpeedSensor )
      { S7_Templates := "time_type := Time" } "TimerAlarm".Mm01SpeedSensorTrip.TON(pt := T#2s, et =>)
      S_Coil( "SafetyAlarms".Mm01SpeedSensorTrip )
   END_RUNG
   RUNG wire#w1
      Contact( "HmiTags".AlarmAck )
      I_Contact( "DiFinal".MMHighSpeedSensor )
      R_Coil( "SafetyAlarms".Mm01SpeedSensorTrip )
   END_RUNG
   // the same network as SCL:
   "TimerAlarm".Mm01SpeedSensorTrip.TON(IN := NOT "AlwaysTRUE" AND "DiFinal".MMHighSpeedSensor, PT := T#2s);
   IF "TimerAlarm".Mm01SpeedSensorTrip.Q THEN "SafetyAlarms".Mm01SpeedSensorTrip := TRUE; END_IF;
   IF NOT "AlwaysTRUE" AND "HmiTags".AlarmAck AND NOT "DiFinal".MMHighSpeedSensor THEN
       "SafetyAlarms".Mm01SpeedSensorTrip := FALSE;
   END_IF;
END_REGION

REGION Network 6: "SafetyAlarms".PowerFailure
   RUNG wire#powerrail
      Contact( "AlwaysTRUE" )
      wire#w1
      Contact( "DiFinal".PowerFailure )
      { S7_Templates := "time_type := Time" } "TimerAlarm".PowerFailure.TON(pt := T#2s, et =>)
      S_Coil( "SafetyAlarms".PowerFailure )
   END_RUNG
   RUNG wire#w1
      Contact( "HmiTags".AlarmAck )
      I_Contact( "DiFinal".PowerFailure )
      R_Coil( "SafetyAlarms".PowerFailure )
   END_RUNG
   // the same network as SCL:
   "TimerAlarm".PowerFailure.TON(IN := "AlwaysTRUE" AND "DiFinal".PowerFailure, PT := T#2s);
   IF "TimerAlarm".PowerFailure.Q THEN "SafetyAlarms".PowerFailure := TRUE; END_IF;
   IF "AlwaysTRUE" AND "HmiTags".AlarmAck AND NOT "DiFinal".PowerFailure THEN
       "SafetyAlarms".PowerFailure := FALSE;
   END_IF;
END_REGION

REGION Network 7: "SafetyAlarms".PlcRestarted
   RUNG wire#powerrail
      I_Contact( "AlwaysTRUE" )
      wire#w1
      Contact( "HmiTags".SystemRestart )
      S_Coil( "SafetyAlarms".PlcRestarted )
   END_RUNG
   RUNG wire#w1
      Contact( "HmiTags".AlarmAck )
      I_Contact( "HmiTags".SystemRestart )
      R_Coil( "SafetyAlarms".PlcRestarted )
   END_RUNG
   // the same network as SCL:
   IF NOT "AlwaysTRUE" AND "HmiTags".SystemRestart THEN "SafetyAlarms".PlcRestarted := TRUE; END_IF;
   IF NOT "AlwaysTRUE" AND "HmiTags".AlarmAck AND NOT "HmiTags".SystemRestart THEN
       "SafetyAlarms".PlcRestarted := FALSE;
   END_IF;
END_REGION

REGION Network 8: "SafetyAlarms".Mm01OverloadTrip
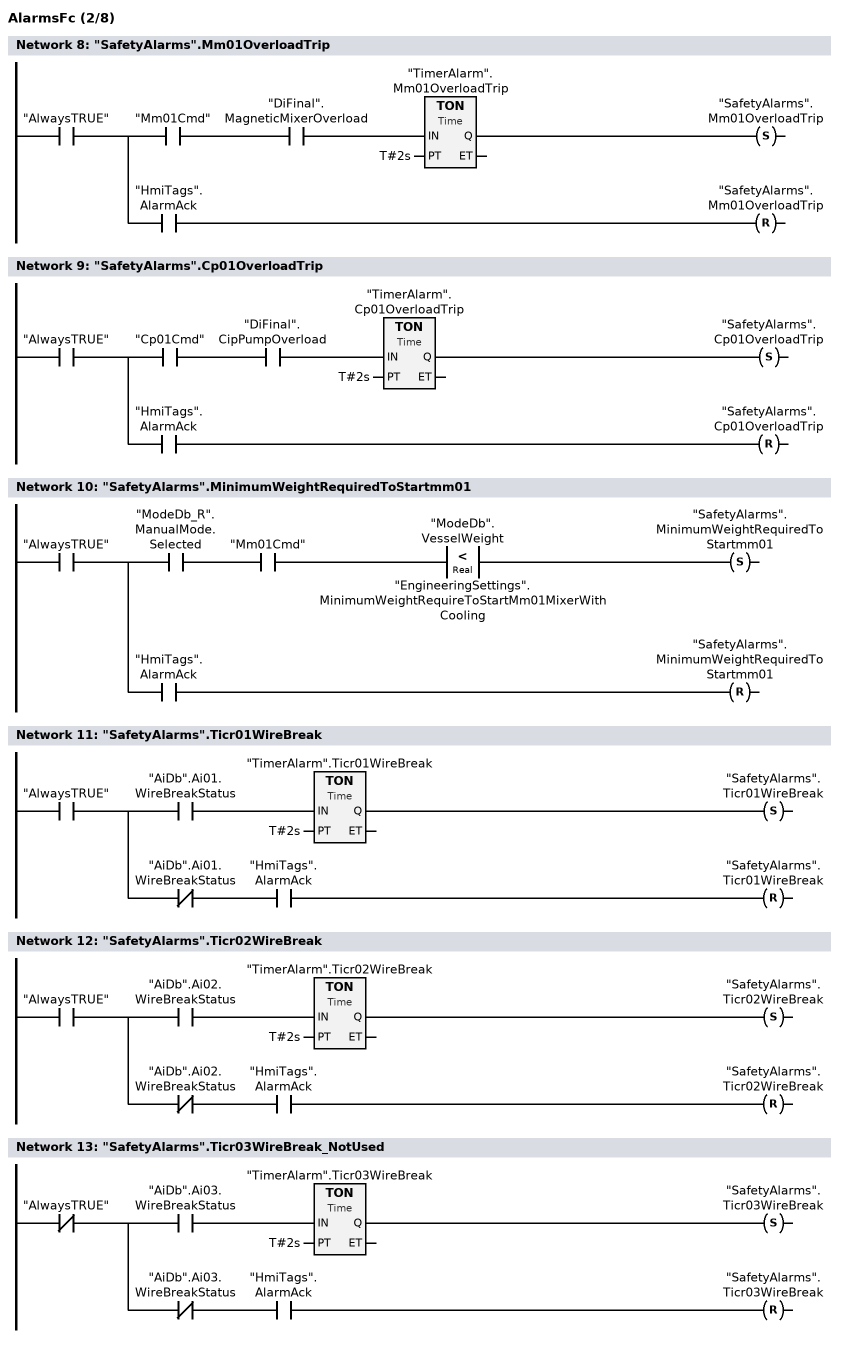
   RUNG wire#powerrail
      Contact( "AlwaysTRUE" )
      wire#w1
      Contact( "Mm01Cmd" )
      Contact( "DiFinal".MagneticMixerOverload )
      { S7_Templates := "time_type := Time" } "TimerAlarm".Mm01OverloadTrip.TON(pt := T#2s, et =>)
      S_Coil( "SafetyAlarms".Mm01OverloadTrip )
   END_RUNG
   RUNG wire#w1
      Contact( "HmiTags".AlarmAck )
      R_Coil( "SafetyAlarms".Mm01OverloadTrip )
   END_RUNG
   // the same network as SCL:
   "TimerAlarm".Mm01OverloadTrip.TON(IN := "AlwaysTRUE" AND "Mm01Cmd" AND "DiFinal".MagneticMixerOverload,
                           PT := T#2s);
   IF "TimerAlarm".Mm01OverloadTrip.Q THEN "SafetyAlarms".Mm01OverloadTrip := TRUE; END_IF;
   IF "AlwaysTRUE" AND "HmiTags".AlarmAck THEN "SafetyAlarms".Mm01OverloadTrip := FALSE; END_IF;
END_REGION

REGION Network 9: "SafetyAlarms".Cp01OverloadTrip
   RUNG wire#powerrail
      Contact( "AlwaysTRUE" )
      wire#w1
      Contact( "Cp01Cmd" )
      Contact( "DiFinal".CipPumpOverload )
      { S7_Templates := "time_type := Time" } "TimerAlarm".Cp01OverloadTrip.TON(pt := T#2s, et =>)
      S_Coil( "SafetyAlarms".Cp01OverloadTrip )
   END_RUNG
   RUNG wire#w1
      Contact( "HmiTags".AlarmAck )
      R_Coil( "SafetyAlarms".Cp01OverloadTrip )
   END_RUNG
   // the same network as SCL:
   "TimerAlarm".Cp01OverloadTrip.TON(IN := "AlwaysTRUE" AND "Cp01Cmd" AND "DiFinal".CipPumpOverload, PT := T#2s);
   IF "TimerAlarm".Cp01OverloadTrip.Q THEN "SafetyAlarms".Cp01OverloadTrip := TRUE; END_IF;
   IF "AlwaysTRUE" AND "HmiTags".AlarmAck THEN "SafetyAlarms".Cp01OverloadTrip := FALSE; END_IF;
END_REGION

REGION Network 10: "SafetyAlarms".MinimumWeightRequiredToStartmm01
   RUNG wire#powerrail
      Contact( "AlwaysTRUE" )
      wire#w1
      Contact( "ModeDb_R".ManualMode.Selected )
      Contact( "Mm01Cmd" )
      { S7_Templates := "SrcType := Real" } LT_Contact(in1 := "ModeDb".VesselWeight, in2 := "EngineeringSettings".MinimumWeightRequireToStartMm01MixerWithCooling)
      S_Coil( "SafetyAlarms".MinimumWeightRequiredToStartmm01 )
   END_RUNG
   RUNG wire#w1
      Contact( "HmiTags".AlarmAck )
      R_Coil( "SafetyAlarms".MinimumWeightRequiredToStartmm01 )
   END_RUNG
   // the same network as SCL:
   IF "AlwaysTRUE" AND "ModeDb_R".ManualMode.Selected AND "Mm01Cmd" AND ("ModeDb".VesselWeight < "EngineeringSettings".MinimumWeightRequireToStartMm01MixerWithCooling) THEN
       "SafetyAlarms".MinimumWeightRequiredToStartmm01 := TRUE;
   END_IF;
   IF "AlwaysTRUE" AND "HmiTags".AlarmAck THEN
       "SafetyAlarms".MinimumWeightRequiredToStartmm01 := FALSE;
   END_IF;
END_REGION

REGION Network 11: "SafetyAlarms".Ticr01WireBreak
   RUNG wire#powerrail
      Contact( "AlwaysTRUE" )
      wire#w1
      Contact( "AiDb".Ai01.WireBreakStatus )
      { S7_Templates := "time_type := Time" } "TimerAlarm".Ticr01WireBreak.TON(pt := T#2s, et =>)
      S_Coil( "SafetyAlarms".Ticr01WireBreak )
   END_RUNG
   RUNG wire#w1
      I_Contact( "AiDb".Ai01.WireBreakStatus )
      Contact( "HmiTags".AlarmAck )
      R_Coil( "SafetyAlarms".Ticr01WireBreak )
   END_RUNG
   // the same network as SCL:
   "TimerAlarm".Ticr01WireBreak.TON(IN := "AlwaysTRUE" AND "AiDb".Ai01.WireBreakStatus, PT := T#2s);
   IF "TimerAlarm".Ticr01WireBreak.Q THEN "SafetyAlarms".Ticr01WireBreak := TRUE; END_IF;
   IF "AlwaysTRUE" AND NOT "AiDb".Ai01.WireBreakStatus AND "HmiTags".AlarmAck THEN
       "SafetyAlarms".Ticr01WireBreak := FALSE;
   END_IF;
END_REGION

REGION Network 12: "SafetyAlarms".Ticr02WireBreak
   RUNG wire#powerrail
      Contact( "AlwaysTRUE" )
      wire#w1
      Contact( "AiDb".Ai02.WireBreakStatus )
      { S7_Templates := "time_type := Time" } "TimerAlarm".Ticr02WireBreak.TON(pt := T#2s, et =>)
      S_Coil( "SafetyAlarms".Ticr02WireBreak )
   END_RUNG
   RUNG wire#w1
      I_Contact( "AiDb".Ai02.WireBreakStatus )
      Contact( "HmiTags".AlarmAck )
      R_Coil( "SafetyAlarms".Ticr02WireBreak )
   END_RUNG
   // the same network as SCL:
   "TimerAlarm".Ticr02WireBreak.TON(IN := "AlwaysTRUE" AND "AiDb".Ai02.WireBreakStatus, PT := T#2s);
   IF "TimerAlarm".Ticr02WireBreak.Q THEN "SafetyAlarms".Ticr02WireBreak := TRUE; END_IF;
   IF "AlwaysTRUE" AND NOT "AiDb".Ai02.WireBreakStatus AND "HmiTags".AlarmAck THEN
       "SafetyAlarms".Ticr02WireBreak := FALSE;
   END_IF;
END_REGION

REGION Network 13: "SafetyAlarms".Ticr03WireBreak_NotUsed
   RUNG wire#powerrail
      I_Contact( "AlwaysTRUE" )
      wire#w1
      Contact( "AiDb".Ai03.WireBreakStatus )
      { S7_Templates := "time_type := Time" } "TimerAlarm".Ticr03WireBreak.TON(pt := T#2s, et =>)
      S_Coil( "SafetyAlarms".Ticr03WireBreak )
   END_RUNG
   RUNG wire#w1
      I_Contact( "AiDb".Ai03.WireBreakStatus )
      Contact( "HmiTags".AlarmAck )
      R_Coil( "SafetyAlarms".Ticr03WireBreak )
   END_RUNG
   // the same network as SCL:
   "TimerAlarm".Ticr03WireBreak.TON(IN := NOT "AlwaysTRUE" AND "AiDb".Ai03.WireBreakStatus, PT := T#2s);
   IF "TimerAlarm".Ticr03WireBreak.Q THEN "SafetyAlarms".Ticr03WireBreak := TRUE; END_IF;
   IF NOT "AlwaysTRUE" AND NOT "AiDb".Ai03.WireBreakStatus AND "HmiTags".AlarmAck THEN
       "SafetyAlarms".Ticr03WireBreak := FALSE;
   END_IF;
END_REGION

REGION Network 14: "SafetyAlarms".Ticr04WireBreak_NotUsed
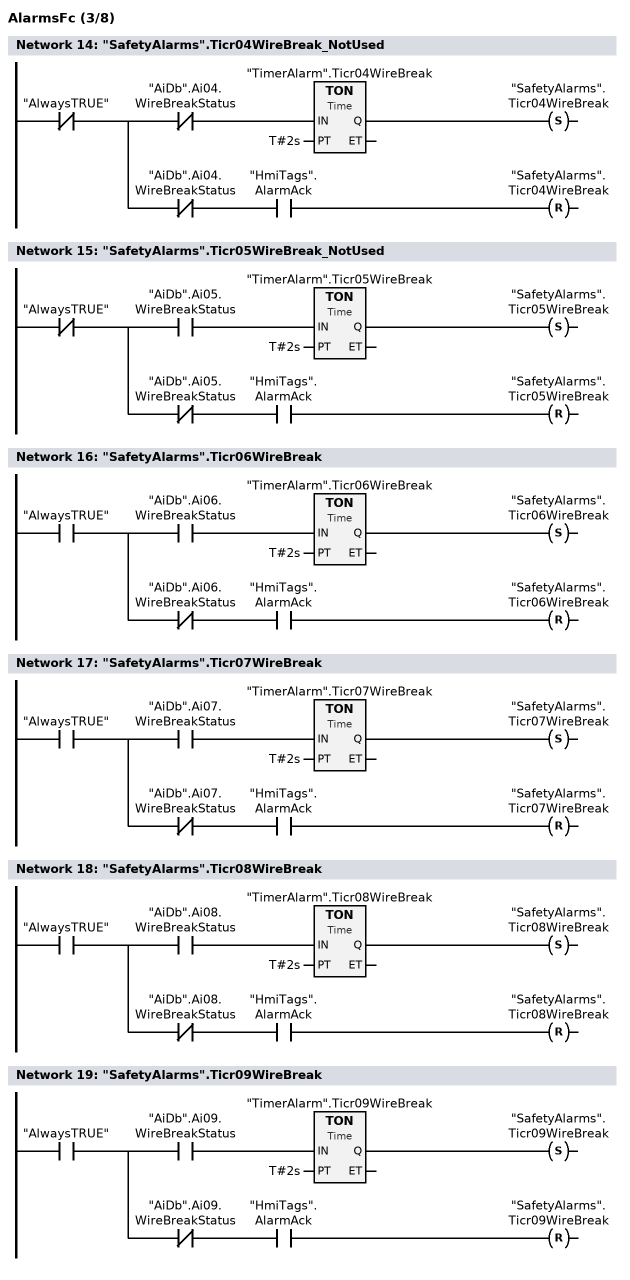
   RUNG wire#powerrail
      I_Contact( "AlwaysTRUE" )
      wire#w1
      I_Contact( "AiDb".Ai04.WireBreakStatus )
      { S7_Templates := "time_type := Time" } "TimerAlarm".Ticr04WireBreak.TON(pt := T#2s, et =>)
      S_Coil( "SafetyAlarms".Ticr04WireBreak )
   END_RUNG
   RUNG wire#w1
      I_Contact( "AiDb".Ai04.WireBreakStatus )
      Contact( "HmiTags".AlarmAck )
      R_Coil( "SafetyAlarms".Ticr04WireBreak )
   END_RUNG
   // the same network as SCL:
   "TimerAlarm".Ticr04WireBreak.TON(IN := NOT "AlwaysTRUE" AND NOT "AiDb".Ai04.WireBreakStatus, PT := T#2s);
   IF "TimerAlarm".Ticr04WireBreak.Q THEN "SafetyAlarms".Ticr04WireBreak := TRUE; END_IF;
   IF NOT "AlwaysTRUE" AND NOT "AiDb".Ai04.WireBreakStatus AND "HmiTags".AlarmAck THEN
       "SafetyAlarms".Ticr04WireBreak := FALSE;
   END_IF;
END_REGION

REGION Network 15: "SafetyAlarms".Ticr05WireBreak_NotUsed
   RUNG wire#powerrail
      I_Contact( "AlwaysTRUE" )
      wire#w1
      Contact( "AiDb".Ai05.WireBreakStatus )
      { S7_Templates := "time_type := Time" } "TimerAlarm".Ticr05WireBreak.TON(pt := T#2s, et =>)
      S_Coil( "SafetyAlarms".Ticr05WireBreak )
   END_RUNG
   RUNG wire#w1
      I_Contact( "AiDb".Ai05.WireBreakStatus )
      Contact( "HmiTags".AlarmAck )
      R_Coil( "SafetyAlarms".Ticr05WireBreak )
   END_RUNG
   // the same network as SCL:
   "TimerAlarm".Ticr05WireBreak.TON(IN := NOT "AlwaysTRUE" AND "AiDb".Ai05.WireBreakStatus, PT := T#2s);
   IF "TimerAlarm".Ticr05WireBreak.Q THEN "SafetyAlarms".Ticr05WireBreak := TRUE; END_IF;
   IF NOT "AlwaysTRUE" AND NOT "AiDb".Ai05.WireBreakStatus AND "HmiTags".AlarmAck THEN
       "SafetyAlarms".Ticr05WireBreak := FALSE;
   END_IF;
END_REGION

REGION Network 16: "SafetyAlarms".Ticr06WireBreak
   RUNG wire#powerrail
      Contact( "AlwaysTRUE" )
      wire#w1
      Contact( "AiDb".Ai06.WireBreakStatus )
      { S7_Templates := "time_type := Time" } "TimerAlarm".Ticr06WireBreak.TON(pt := T#2s, et =>)
      S_Coil( "SafetyAlarms".Ticr06WireBreak )
   END_RUNG
   RUNG wire#w1
      I_Contact( "AiDb".Ai06.WireBreakStatus )
      Contact( "HmiTags".AlarmAck )
      R_Coil( "SafetyAlarms".Ticr06WireBreak )
   END_RUNG
   // the same network as SCL:
   "TimerAlarm".Ticr06WireBreak.TON(IN := "AlwaysTRUE" AND "AiDb".Ai06.WireBreakStatus, PT := T#2s);
   IF "TimerAlarm".Ticr06WireBreak.Q THEN "SafetyAlarms".Ticr06WireBreak := TRUE; END_IF;
   IF "AlwaysTRUE" AND NOT "AiDb".Ai06.WireBreakStatus AND "HmiTags".AlarmAck THEN
       "SafetyAlarms".Ticr06WireBreak := FALSE;
   END_IF;
END_REGION

REGION Network 17: "SafetyAlarms".Ticr07WireBreak
   RUNG wire#powerrail
      Contact( "AlwaysTRUE" )
      wire#w1
      Contact( "AiDb".Ai07.WireBreakStatus )
      { S7_Templates := "time_type := Time" } "TimerAlarm".Ticr07WireBreak.TON(pt := T#2s, et =>)
      S_Coil( "SafetyAlarms".Ticr07WireBreak )
   END_RUNG
   RUNG wire#w1
      I_Contact( "AiDb".Ai07.WireBreakStatus )
      Contact( "HmiTags".AlarmAck )
      R_Coil( "SafetyAlarms".Ticr07WireBreak )
   END_RUNG
   // the same network as SCL:
   "TimerAlarm".Ticr07WireBreak.TON(IN := "AlwaysTRUE" AND "AiDb".Ai07.WireBreakStatus, PT := T#2s);
   IF "TimerAlarm".Ticr07WireBreak.Q THEN "SafetyAlarms".Ticr07WireBreak := TRUE; END_IF;
   IF "AlwaysTRUE" AND NOT "AiDb".Ai07.WireBreakStatus AND "HmiTags".AlarmAck THEN
       "SafetyAlarms".Ticr07WireBreak := FALSE;
   END_IF;
END_REGION

REGION Network 18: "SafetyAlarms".Ticr08WireBreak
   RUNG wire#powerrail
      Contact( "AlwaysTRUE" )
      wire#w1
      Contact( "AiDb".Ai08.WireBreakStatus )
      { S7_Templates := "time_type := Time" } "TimerAlarm".Ticr08WireBreak.TON(pt := T#2s, et =>)
      S_Coil( "SafetyAlarms".Ticr08WireBreak )
   END_RUNG
   RUNG wire#w1
      I_Contact( "AiDb".Ai08.WireBreakStatus )
      Contact( "HmiTags".AlarmAck )
      R_Coil( "SafetyAlarms".Ticr08WireBreak )
   END_RUNG
   // the same network as SCL:
   "TimerAlarm".Ticr08WireBreak.TON(IN := "AlwaysTRUE" AND "AiDb".Ai08.WireBreakStatus, PT := T#2s);
   IF "TimerAlarm".Ticr08WireBreak.Q THEN "SafetyAlarms".Ticr08WireBreak := TRUE; END_IF;
   IF "AlwaysTRUE" AND NOT "AiDb".Ai08.WireBreakStatus AND "HmiTags".AlarmAck THEN
       "SafetyAlarms".Ticr08WireBreak := FALSE;
   END_IF;
END_REGION

REGION Network 19: "SafetyAlarms".Ticr09WireBreak
   RUNG wire#powerrail
      Contact( "AlwaysTRUE" )
      wire#w1
      Contact( "AiDb".Ai09.WireBreakStatus )
      { S7_Templates := "time_type := Time" } "TimerAlarm".Ticr09WireBreak.TON(pt := T#2s, et =>)
      S_Coil( "SafetyAlarms".Ticr09WireBreak )
   END_RUNG
   RUNG wire#w1
      I_Contact( "AiDb".Ai09.WireBreakStatus )
      Contact( "HmiTags".AlarmAck )
      R_Coil( "SafetyAlarms".Ticr09WireBreak )
   END_RUNG
   // the same network as SCL:
   "TimerAlarm".Ticr09WireBreak.TON(IN := "AlwaysTRUE" AND "AiDb".Ai09.WireBreakStatus, PT := T#2s);
   IF "TimerAlarm".Ticr09WireBreak.Q THEN "SafetyAlarms".Ticr09WireBreak := TRUE; END_IF;
   IF "AlwaysTRUE" AND NOT "AiDb".Ai09.WireBreakStatus AND "HmiTags".AlarmAck THEN
       "SafetyAlarms".Ticr09WireBreak := FALSE;
   END_IF;
END_REGION

REGION Network 20: "SafetyAlarms".Ticr10WireBreak
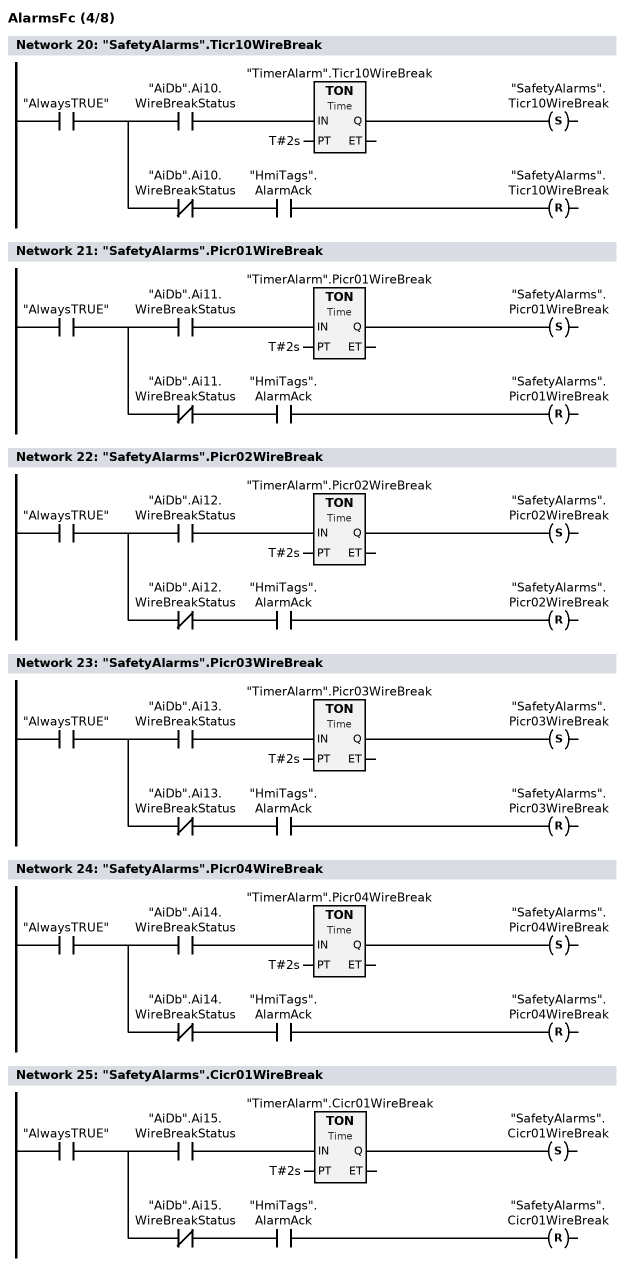
   RUNG wire#powerrail
      Contact( "AlwaysTRUE" )
      wire#w1
      Contact( "AiDb".Ai10.WireBreakStatus )
      { S7_Templates := "time_type := Time" } "TimerAlarm".Ticr10WireBreak.TON(pt := T#2s, et =>)
      S_Coil( "SafetyAlarms".Ticr10WireBreak )
   END_RUNG
   RUNG wire#w1
      I_Contact( "AiDb".Ai10.WireBreakStatus )
      Contact( "HmiTags".AlarmAck )
      R_Coil( "SafetyAlarms".Ticr10WireBreak )
   END_RUNG
   // the same network as SCL:
   "TimerAlarm".Ticr10WireBreak.TON(IN := "AlwaysTRUE" AND "AiDb".Ai10.WireBreakStatus, PT := T#2s);
   IF "TimerAlarm".Ticr10WireBreak.Q THEN "SafetyAlarms".Ticr10WireBreak := TRUE; END_IF;
   IF "AlwaysTRUE" AND NOT "AiDb".Ai10.WireBreakStatus AND "HmiTags".AlarmAck THEN
       "SafetyAlarms".Ticr10WireBreak := FALSE;
   END_IF;
END_REGION

REGION Network 21: "SafetyAlarms".Picr01WireBreak
   RUNG wire#powerrail
      Contact( "AlwaysTRUE" )
      wire#w1
      Contact( "AiDb".Ai11.WireBreakStatus )
      { S7_Templates := "time_type := Time" } "TimerAlarm".Picr01WireBreak.TON(pt := T#2s, et =>)
      S_Coil( "SafetyAlarms".Picr01WireBreak )
   END_RUNG
   RUNG wire#w1
      I_Contact( "AiDb".Ai11.WireBreakStatus )
      Contact( "HmiTags".AlarmAck )
      R_Coil( "SafetyAlarms".Picr01WireBreak )
   END_RUNG
   // the same network as SCL:
   "TimerAlarm".Picr01WireBreak.TON(IN := "AlwaysTRUE" AND "AiDb".Ai11.WireBreakStatus, PT := T#2s);
   IF "TimerAlarm".Picr01WireBreak.Q THEN "SafetyAlarms".Picr01WireBreak := TRUE; END_IF;
   IF "AlwaysTRUE" AND NOT "AiDb".Ai11.WireBreakStatus AND "HmiTags".AlarmAck THEN
       "SafetyAlarms".Picr01WireBreak := FALSE;
   END_IF;
END_REGION

REGION Network 22: "SafetyAlarms".Picr02WireBreak
   RUNG wire#powerrail
      Contact( "AlwaysTRUE" )
      wire#w1
      Contact( "AiDb".Ai12.WireBreakStatus )
      { S7_Templates := "time_type := Time" } "TimerAlarm".Picr02WireBreak.TON(pt := T#2s, et =>)
      S_Coil( "SafetyAlarms".Picr02WireBreak )
   END_RUNG
   RUNG wire#w1
      I_Contact( "AiDb".Ai12.WireBreakStatus )
      Contact( "HmiTags".AlarmAck )
      R_Coil( "SafetyAlarms".Picr02WireBreak )
   END_RUNG
   // the same network as SCL:
   "TimerAlarm".Picr02WireBreak.TON(IN := "AlwaysTRUE" AND "AiDb".Ai12.WireBreakStatus, PT := T#2s);
   IF "TimerAlarm".Picr02WireBreak.Q THEN "SafetyAlarms".Picr02WireBreak := TRUE; END_IF;
   IF "AlwaysTRUE" AND NOT "AiDb".Ai12.WireBreakStatus AND "HmiTags".AlarmAck THEN
       "SafetyAlarms".Picr02WireBreak := FALSE;
   END_IF;
END_REGION

REGION Network 23: "SafetyAlarms".Picr03WireBreak
   RUNG wire#powerrail
      Contact( "AlwaysTRUE" )
      wire#w1
      Contact( "AiDb".Ai13.WireBreakStatus )
      { S7_Templates := "time_type := Time" } "TimerAlarm".Picr03WireBreak.TON(pt := T#2s, et =>)
      S_Coil( "SafetyAlarms".Picr03WireBreak )
   END_RUNG
   RUNG wire#w1
      I_Contact( "AiDb".Ai13.WireBreakStatus )
      Contact( "HmiTags".AlarmAck )
      R_Coil( "SafetyAlarms".Picr03WireBreak )
   END_RUNG
   // the same network as SCL:
   "TimerAlarm".Picr03WireBreak.TON(IN := "AlwaysTRUE" AND "AiDb".Ai13.WireBreakStatus, PT := T#2s);
   IF "TimerAlarm".Picr03WireBreak.Q THEN "SafetyAlarms".Picr03WireBreak := TRUE; END_IF;
   IF "AlwaysTRUE" AND NOT "AiDb".Ai13.WireBreakStatus AND "HmiTags".AlarmAck THEN
       "SafetyAlarms".Picr03WireBreak := FALSE;
   END_IF;
END_REGION

REGION Network 24: "SafetyAlarms".Picr04WireBreak
   RUNG wire#powerrail
      Contact( "AlwaysTRUE" )
      wire#w1
      Contact( "AiDb".Ai14.WireBreakStatus )
      { S7_Templates := "time_type := Time" } "TimerAlarm".Picr04WireBreak.TON(pt := T#2s, et =>)
      S_Coil( "SafetyAlarms".Picr04WireBreak )
   END_RUNG
   RUNG wire#w1
      I_Contact( "AiDb".Ai14.WireBreakStatus )
      Contact( "HmiTags".AlarmAck )
      R_Coil( "SafetyAlarms".Picr04WireBreak )
   END_RUNG
   // the same network as SCL:
   "TimerAlarm".Picr04WireBreak.TON(IN := "AlwaysTRUE" AND "AiDb".Ai14.WireBreakStatus, PT := T#2s);
   IF "TimerAlarm".Picr04WireBreak.Q THEN "SafetyAlarms".Picr04WireBreak := TRUE; END_IF;
   IF "AlwaysTRUE" AND NOT "AiDb".Ai14.WireBreakStatus AND "HmiTags".AlarmAck THEN
       "SafetyAlarms".Picr04WireBreak := FALSE;
   END_IF;
END_REGION

REGION Network 25: "SafetyAlarms".Cicr01WireBreak
   RUNG wire#powerrail
      Contact( "AlwaysTRUE" )
      wire#w1
      Contact( "AiDb".Ai15.WireBreakStatus )
      { S7_Templates := "time_type := Time" } "TimerAlarm".Cicr01WireBreak.TON(pt := T#2s, et =>)
      S_Coil( "SafetyAlarms".Cicr01WireBreak )
   END_RUNG
   RUNG wire#w1
      I_Contact( "AiDb".Ai15.WireBreakStatus )
      Contact( "HmiTags".AlarmAck )
      R_Coil( "SafetyAlarms".Cicr01WireBreak )
   END_RUNG
   // the same network as SCL:
   "TimerAlarm".Cicr01WireBreak.TON(IN := "AlwaysTRUE" AND "AiDb".Ai15.WireBreakStatus, PT := T#2s);
   IF "TimerAlarm".Cicr01WireBreak.Q THEN "SafetyAlarms".Cicr01WireBreak := TRUE; END_IF;
   IF "AlwaysTRUE" AND NOT "AiDb".Ai15.WireBreakStatus AND "HmiTags".AlarmAck THEN
       "SafetyAlarms".Cicr01WireBreak := FALSE;
   END_IF;
END_REGION

REGION Network 26: "SafetyAlarms".Lc01CommunicationFailed
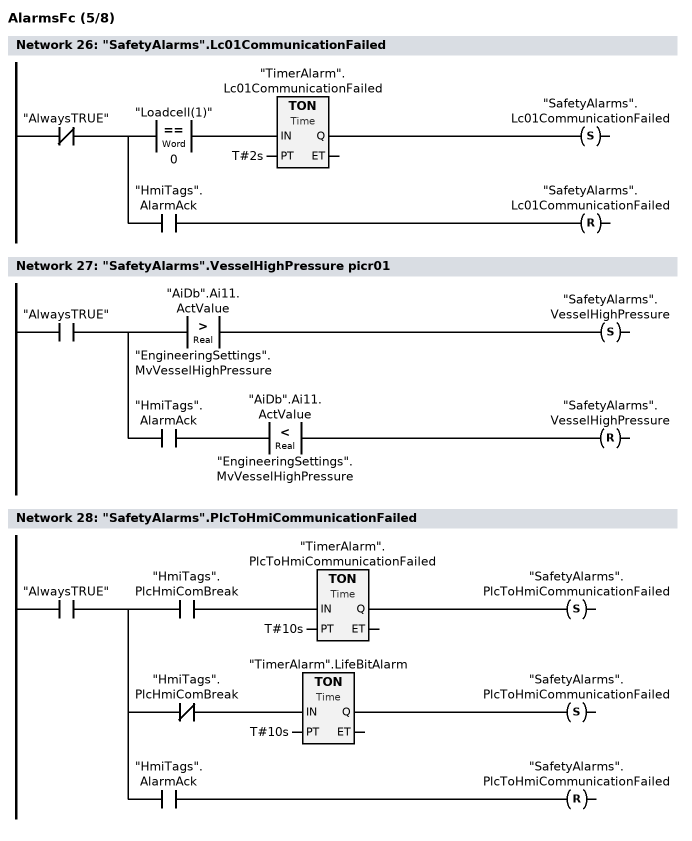
   RUNG wire#powerrail
      I_Contact( "AlwaysTRUE" )
      wire#w1
      { S7_Templates := "SrcType := Word" } EQ_Contact(in1 := "Loadcell(1)", in2 := 0)
      { S7_Templates := "time_type := Time" } "TimerAlarm".Lc01CommunicationFailed.TON(pt := T#2s, et =>)
      S_Coil( "SafetyAlarms".Lc01CommunicationFailed )
   END_RUNG
   RUNG wire#w1
      Contact( "HmiTags".AlarmAck )
      R_Coil( "SafetyAlarms".Lc01CommunicationFailed )
   END_RUNG
   // the same network as SCL:
   "TimerAlarm".Lc01CommunicationFailed.TON(IN := NOT "AlwaysTRUE" AND ("Loadcell(1)" = 0), PT := T#2s);
   IF "TimerAlarm".Lc01CommunicationFailed.Q THEN "SafetyAlarms".Lc01CommunicationFailed := TRUE; END_IF;
   IF NOT "AlwaysTRUE" AND "HmiTags".AlarmAck THEN "SafetyAlarms".Lc01CommunicationFailed := FALSE; END_IF;
END_REGION

REGION Network 27: "SafetyAlarms".VesselHighPressure picr01
   RUNG wire#powerrail
      Contact( "AlwaysTRUE" )
      wire#w1
      { S7_Templates := "SrcType := Real" } GT_Contact(in1 := "AiDb".Ai11.ActValue, in2 := "EngineeringSettings".MvVesselHighPressure)
      S_Coil( "SafetyAlarms".VesselHighPressure )
   END_RUNG
   RUNG wire#w1
      Contact( "HmiTags".AlarmAck )
      { S7_Templates := "SrcType := Real" } LT_Contact(in1 := "AiDb".Ai11.ActValue, in2 := "EngineeringSettings".MvVesselHighPressure)
      R_Coil( "SafetyAlarms".VesselHighPressure )
   END_RUNG
   // the same network as SCL:
   IF "AlwaysTRUE" AND ("AiDb".Ai11.ActValue > "EngineeringSettings".MvVesselHighPressure) THEN
       "SafetyAlarms".VesselHighPressure := TRUE;
   END_IF;
   IF "AlwaysTRUE" AND "HmiTags".AlarmAck AND ("AiDb".Ai11.ActValue < "EngineeringSettings".MvVesselHighPressure) THEN
       "SafetyAlarms".VesselHighPressure := FALSE;
   END_IF;
END_REGION

REGION Network 28: "SafetyAlarms".PlcToHmiCommunicationFailed
   RUNG wire#powerrail
      Contact( "AlwaysTRUE" )
      wire#w1
      Contact( "HmiTags".PlcHmiComBreak )
      { S7_Templates := "time_type := Time" } "TimerAlarm".PlcToHmiCommunicationFailed.TON(pt := T#10s, et =>)
      S_Coil( "SafetyAlarms".PlcToHmiCommunicationFailed )
   END_RUNG
   RUNG wire#w1
      I_Contact( "HmiTags".PlcHmiComBreak )
      { S7_Templates := "time_type := Time" } "TimerAlarm".LifeBitAlarm.TON(pt := T#10s, et =>)
      S_Coil( "SafetyAlarms".PlcToHmiCommunicationFailed )
   END_RUNG
   RUNG wire#w1
      Contact( "HmiTags".AlarmAck )
      R_Coil( "SafetyAlarms".PlcToHmiCommunicationFailed )
   END_RUNG
   // the same network as SCL:
   "TimerAlarm".PlcToHmiCommunicationFailed.TON(IN := "AlwaysTRUE" AND "HmiTags".PlcHmiComBreak, PT := T#10s);
   IF "TimerAlarm".PlcToHmiCommunicationFailed.Q THEN
       "SafetyAlarms".PlcToHmiCommunicationFailed := TRUE;
   END_IF;
   "TimerAlarm".LifeBitAlarm.TON(IN := "AlwaysTRUE" AND NOT "HmiTags".PlcHmiComBreak, PT := T#10s);
   IF "TimerAlarm".LifeBitAlarm.Q THEN "SafetyAlarms".PlcToHmiCommunicationFailed := TRUE; END_IF;
   IF "AlwaysTRUE" AND "HmiTags".AlarmAck THEN "SafetyAlarms".PlcToHmiCommunicationFailed := FALSE; END_IF;
END_REGION

REGION Network 29: "HmiTags".ManualModeFAULT
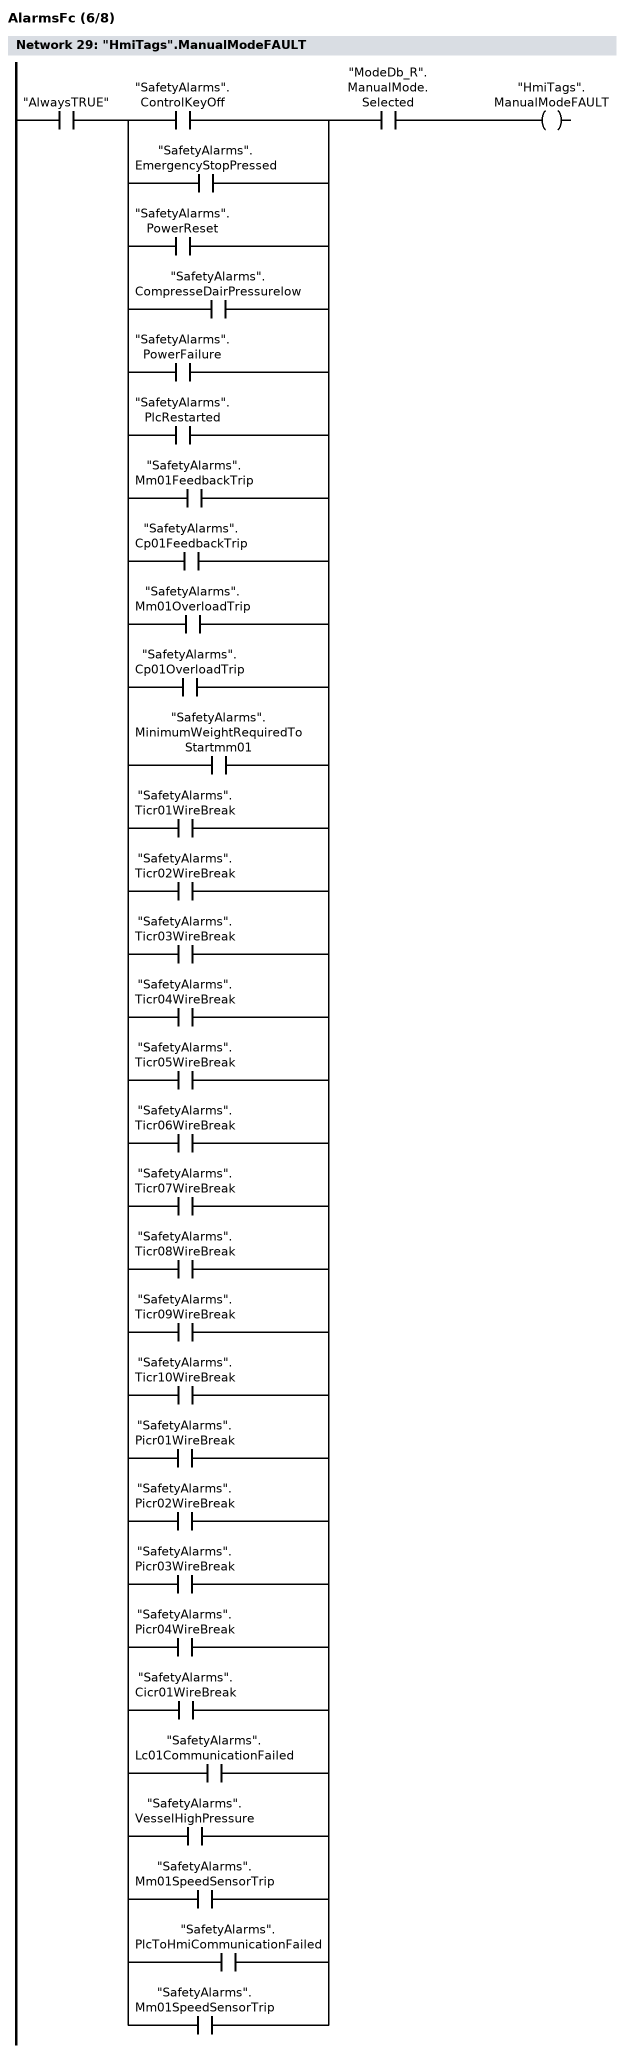
   RUNG wire#powerrail
      Contact( "AlwaysTRUE" )
      wire#w1
      Contact( "SafetyAlarms".ControlKeyOff )
      wire#w2
      Contact( "ModeDb_R".ManualMode.Selected )
      Coil( "HmiTags".ManualModeFAULT )
   END_RUNG
   RUNG wire#w1
      Contact( "SafetyAlarms".EmergencyStopPressed )
   END_RUNG wire#w2
   RUNG wire#w1
      Contact( "SafetyAlarms".PowerReset )
   END_RUNG wire#w2
   RUNG wire#w1
      Contact( "SafetyAlarms".CompresseDairPressurelow )
   END_RUNG wire#w2
   RUNG wire#w1
      Contact( "SafetyAlarms".PowerFailure )
   END_RUNG wire#w2
   RUNG wire#w1
      Contact( "SafetyAlarms".PlcRestarted )
   END_RUNG wire#w2
   RUNG wire#w1
      Contact( "SafetyAlarms".Mm01FeedbackTrip )
   END_RUNG wire#w2
   RUNG wire#w1
      Contact( "SafetyAlarms".Cp01FeedbackTrip )
   END_RUNG wire#w2
   RUNG wire#w1
      Contact( "SafetyAlarms".Mm01OverloadTrip )
   END_RUNG wire#w2
   RUNG wire#w1
      Contact( "SafetyAlarms".Cp01OverloadTrip )
   END_RUNG wire#w2
   RUNG wire#w1
      Contact( "SafetyAlarms".MinimumWeightRequiredToStartmm01 )
   END_RUNG wire#w2
   RUNG wire#w1
      Contact( "SafetyAlarms".Ticr01WireBreak )
   END_RUNG wire#w2
   RUNG wire#w1
      Contact( "SafetyAlarms".Ticr02WireBreak )
   END_RUNG wire#w2
   RUNG wire#w1
      Contact( "SafetyAlarms".Ticr03WireBreak )
   END_RUNG wire#w2
   RUNG wire#w1
      Contact( "SafetyAlarms".Ticr04WireBreak )
   END_RUNG wire#w2
   RUNG wire#w1
      Contact( "SafetyAlarms".Ticr05WireBreak )
   END_RUNG wire#w2
   RUNG wire#w1
      Contact( "SafetyAlarms".Ticr06WireBreak )
   END_RUNG wire#w2
   RUNG wire#w1
      Contact( "SafetyAlarms".Ticr07WireBreak )
   END_RUNG wire#w2
   RUNG wire#w1
      Contact( "SafetyAlarms".Ticr08WireBreak )
   END_RUNG wire#w2
   RUNG wire#w1
      Contact( "SafetyAlarms".Ticr09WireBreak )
   END_RUNG wire#w2
   RUNG wire#w1
      Contact( "SafetyAlarms".Ticr10WireBreak )
   END_RUNG wire#w2
   RUNG wire#w1
      Contact( "SafetyAlarms".Picr01WireBreak )
   END_RUNG wire#w2
   RUNG wire#w1
      Contact( "SafetyAlarms".Picr02WireBreak )
   END_RUNG wire#w2
   RUNG wire#w1
      Contact( "SafetyAlarms".Picr03WireBreak )
   END_RUNG wire#w2
   RUNG wire#w1
      Contact( "SafetyAlarms".Picr04WireBreak )
   END_RUNG wire#w2
   RUNG wire#w1
      Contact( "SafetyAlarms".Cicr01WireBreak )
   END_RUNG wire#w2
   RUNG wire#w1
      Contact( "SafetyAlarms".Lc01CommunicationFailed )
   END_RUNG wire#w2
   RUNG wire#w1
      Contact( "SafetyAlarms".VesselHighPressure )
   END_RUNG wire#w2
   RUNG wire#w1
      Contact( "SafetyAlarms".Mm01SpeedSensorTrip )
   END_RUNG wire#w2
   RUNG wire#w1
      Contact( "SafetyAlarms".PlcToHmiCommunicationFailed )
   END_RUNG wire#w2
   RUNG wire#w1
      Contact( "SafetyAlarms".Mm01SpeedSensorTrip )
   END_RUNG wire#w2
   // the same network as SCL:
   "HmiTags".ManualModeFAULT := "AlwaysTRUE" AND ("SafetyAlarms".ControlKeyOff OR "SafetyAlarms".EmergencyStopPressed OR "SafetyAlarms".PowerReset OR "SafetyAlarms".CompresseDairPressurelow OR "SafetyAlarms".PowerFailure OR "SafetyAlarms".PlcRestarted OR "SafetyAlarms".Mm01FeedbackTrip OR "SafetyAlarms".Cp01FeedbackTrip OR "SafetyAlarms".Mm01OverloadTrip OR "SafetyAlarms".Cp01OverloadTrip OR "SafetyAlarms".MinimumWeightRequiredToStartmm01 OR "SafetyAlarms".Ticr01WireBreak OR "SafetyAlarms".Ticr02WireBreak OR "SafetyAlarms".Ticr03WireBreak OR "SafetyAlarms".Ticr04WireBreak OR "SafetyAlarms".Ticr05WireBreak OR "SafetyAlarms".Ticr06WireBreak OR "SafetyAlarms".Ticr07WireBreak OR "SafetyAlarms".Ticr08WireBreak OR "SafetyAlarms".Ticr09WireBreak OR "SafetyAlarms".Ticr10WireBreak OR "SafetyAlarms".Picr01WireBreak OR "SafetyAlarms".Picr02WireBreak OR "SafetyAlarms".Picr03WireBreak OR "SafetyAlarms".Picr04WireBreak OR "SafetyAlarms".Cicr01WireBreak OR "SafetyAlarms".Lc01CommunicationFailed OR "SafetyAlarms".VesselHighPressure OR "SafetyAlarms".Mm01SpeedSensorTrip OR "SafetyAlarms".PlcToHmiCommunicationFailed OR "SafetyAlarms".Mm01SpeedSensorTrip) AND "ModeDb_R".ManualMode.Selected;
END_REGION

REGION Network 30: "HmiTags".Hooter -- set
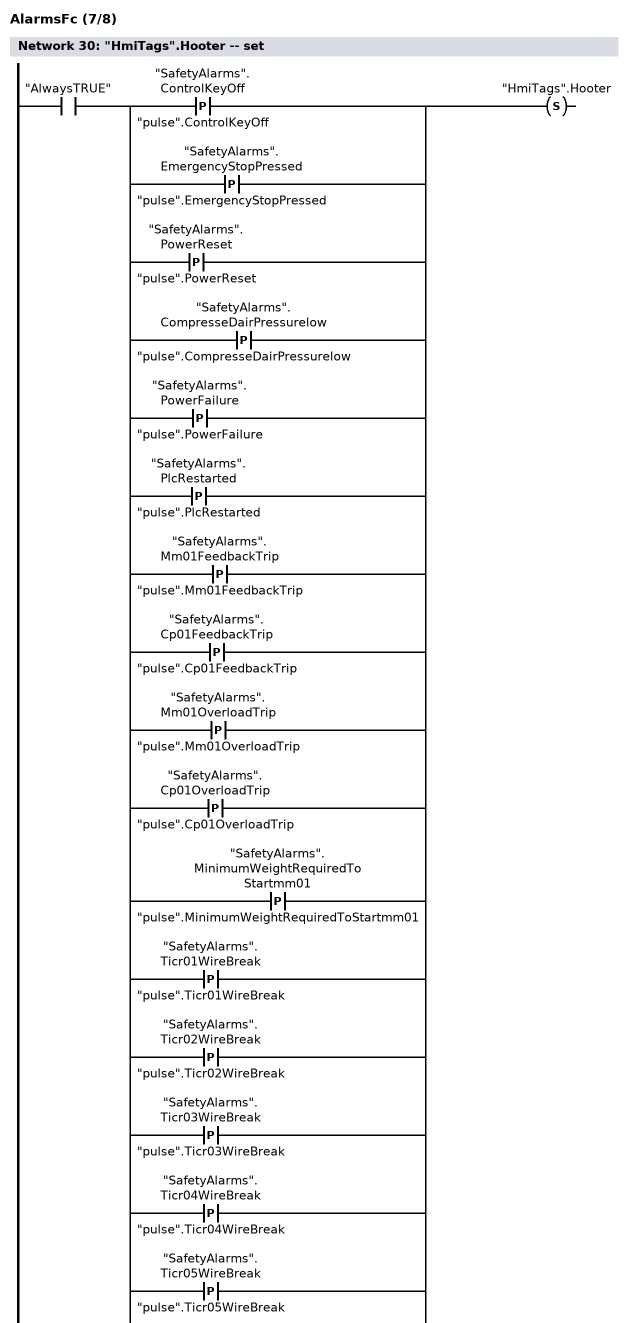
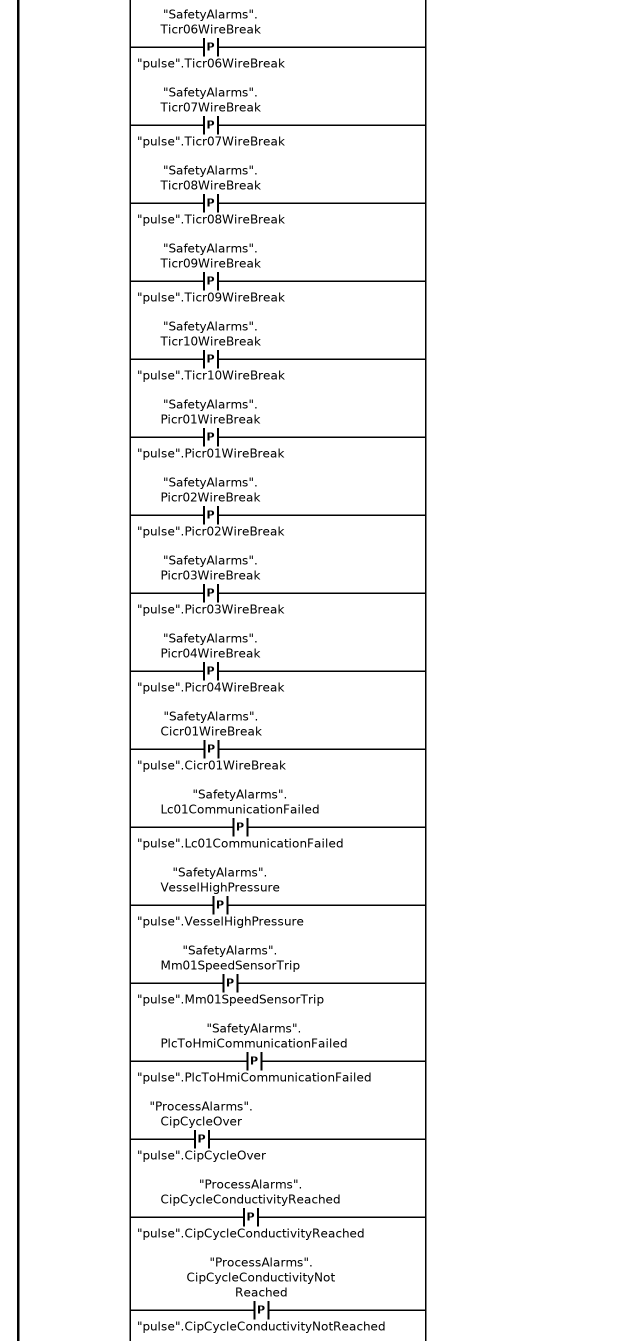
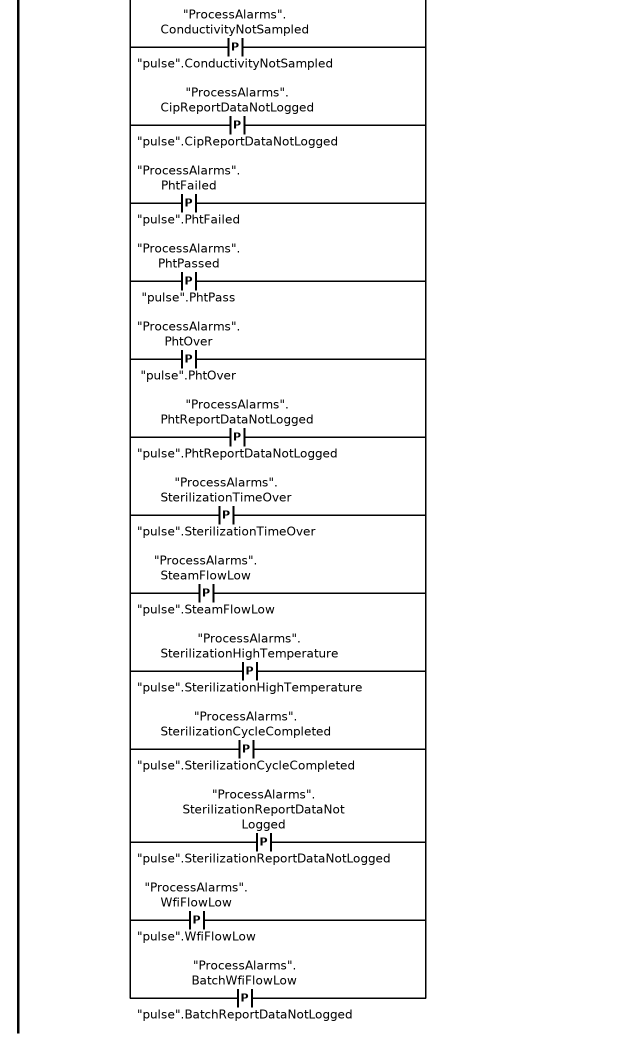
   RUNG wire#powerrail
      Contact( "AlwaysTRUE" )
      wire#w1
      P_Contact(operand := "SafetyAlarms".ControlKeyOff, bit := "pulse".ControlKeyOff)
      wire#w2
      S_Coil( "HmiTags".Hooter )
   END_RUNG
   RUNG wire#w1
      P_Contact(operand := "SafetyAlarms".EmergencyStopPressed, bit := "pulse".EmergencyStopPressed)
   END_RUNG wire#w2
   RUNG wire#w1
      P_Contact(operand := "SafetyAlarms".PowerReset, bit := "pulse".PowerReset)
   END_RUNG wire#w2
   RUNG wire#w1
      P_Contact(operand := "SafetyAlarms".CompresseDairPressurelow, bit := "pulse".CompresseDairPressurelow)
   END_RUNG wire#w2
   RUNG wire#w1
      P_Contact(operand := "SafetyAlarms".PowerFailure, bit := "pulse".PowerFailure)
   END_RUNG wire#w2
   RUNG wire#w1
      P_Contact(operand := "SafetyAlarms".PlcRestarted, bit := "pulse".PlcRestarted)
   END_RUNG wire#w2
   RUNG wire#w1
      P_Contact(operand := "SafetyAlarms".Mm01FeedbackTrip, bit := "pulse".Mm01FeedbackTrip)
   END_RUNG wire#w2
   RUNG wire#w1
      P_Contact(operand := "SafetyAlarms".Cp01FeedbackTrip, bit := "pulse".Cp01FeedbackTrip)
   END_RUNG wire#w2
   RUNG wire#w1
      P_Contact(operand := "SafetyAlarms".Mm01OverloadTrip, bit := "pulse".Mm01OverloadTrip)
   END_RUNG wire#w2
   RUNG wire#w1
      P_Contact(operand := "SafetyAlarms".Cp01OverloadTrip, bit := "pulse".Cp01OverloadTrip)
   END_RUNG wire#w2
   RUNG wire#w1
      P_Contact(operand := "SafetyAlarms".MinimumWeightRequiredToStartmm01, bit := "pulse".MinimumWeightRequiredToStartmm01)
   END_RUNG wire#w2
   RUNG wire#w1
      P_Contact(operand := "SafetyAlarms".Ticr01WireBreak, bit := "pulse".Ticr01WireBreak)
   END_RUNG wire#w2
   RUNG wire#w1
      P_Contact(operand := "SafetyAlarms".Ticr02WireBreak, bit := "pulse".Ticr02WireBreak)
   END_RUNG wire#w2
   RUNG wire#w1
      P_Contact(operand := "SafetyAlarms".Ticr03WireBreak, bit := "pulse".Ticr03WireBreak)
   END_RUNG wire#w2
   RUNG wire#w1
      P_Contact(operand := "SafetyAlarms".Ticr04WireBreak, bit := "pulse".Ticr04WireBreak)
   END_RUNG wire#w2
   RUNG wire#w1
      P_Contact(operand := "SafetyAlarms".Ticr05WireBreak, bit := "pulse".Ticr05WireBreak)
   END_RUNG wire#w2
   RUNG wire#w1
      P_Contact(operand := "SafetyAlarms".Ticr06WireBreak, bit := "pulse".Ticr06WireBreak)
   END_RUNG wire#w2
   RUNG wire#w1
      P_Contact(operand := "SafetyAlarms".Ticr07WireBreak, bit := "pulse".Ticr07WireBreak)
   END_RUNG wire#w2
   RUNG wire#w1
      P_Contact(operand := "SafetyAlarms".Ticr08WireBreak, bit := "pulse".Ticr08WireBreak)
   END_RUNG wire#w2
   RUNG wire#w1
      P_Contact(operand := "SafetyAlarms".Ticr09WireBreak, bit := "pulse".Ticr09WireBreak)
   END_RUNG wire#w2
   RUNG wire#w1
      P_Contact(operand := "SafetyAlarms".Ticr10WireBreak, bit := "pulse".Ticr10WireBreak)
   END_RUNG wire#w2
   RUNG wire#w1
      P_Contact(operand := "SafetyAlarms".Picr01WireBreak, bit := "pulse".Picr01WireBreak)
   END_RUNG wire#w2
   RUNG wire#w1
      P_Contact(operand := "SafetyAlarms".Picr02WireBreak, bit := "pulse".Picr02WireBreak)
   END_RUNG wire#w2
   RUNG wire#w1
      P_Contact(operand := "SafetyAlarms".Picr03WireBreak, bit := "pulse".Picr03WireBreak)
   END_RUNG wire#w2
   RUNG wire#w1
      P_Contact(operand := "SafetyAlarms".Picr04WireBreak, bit := "pulse".Picr04WireBreak)
   END_RUNG wire#w2
   RUNG wire#w1
      P_Contact(operand := "SafetyAlarms".Cicr01WireBreak, bit := "pulse".Cicr01WireBreak)
   END_RUNG wire#w2
   RUNG wire#w1
      P_Contact(operand := "SafetyAlarms".Lc01CommunicationFailed, bit := "pulse".Lc01CommunicationFailed)
   END_RUNG wire#w2
   RUNG wire#w1
      P_Contact(operand := "SafetyAlarms".VesselHighPressure, bit := "pulse".VesselHighPressure)
   END_RUNG wire#w2
   RUNG wire#w1
      P_Contact(operand := "SafetyAlarms".Mm01SpeedSensorTrip, bit := "pulse".Mm01SpeedSensorTrip)
   END_RUNG wire#w2
   RUNG wire#w1
      P_Contact(operand := "SafetyAlarms".PlcToHmiCommunicationFailed, bit := "pulse".PlcToHmiCommunicationFailed)
   END_RUNG wire#w2
   RUNG wire#w1
      P_Contact(operand := "ProcessAlarms".CipCycleOver, bit := "pulse".CipCycleOver)
   END_RUNG wire#w2
   RUNG wire#w1
      P_Contact(operand := "ProcessAlarms".CipCycleConductivityReached, bit := "pulse".CipCycleConductivityReached)
   END_RUNG wire#w2
   RUNG wire#w1
      P_Contact(operand := "ProcessAlarms".CipCycleConductivityNotReached, bit := "pulse".CipCycleConductivityNotReached)
   END_RUNG wire#w2
   RUNG wire#w1
      P_Contact(operand := "ProcessAlarms".ConductivityNotSampled, bit := "pulse".ConductivityNotSampled)
   END_RUNG wire#w2
   RUNG wire#w1
      P_Contact(operand := "ProcessAlarms".CipReportDataNotLogged, bit := "pulse".CipReportDataNotLogged)
   END_RUNG wire#w2
   RUNG wire#w1
      P_Contact(operand := "ProcessAlarms".PhtFailed, bit := "pulse".PhtFailed)
   END_RUNG wire#w2
   RUNG wire#w1
      P_Contact(operand := "ProcessAlarms".PhtPassed, bit := "pulse".PhtPass)
   END_RUNG wire#w2
   RUNG wire#w1
      P_Contact(operand := "ProcessAlarms".PhtOver, bit := "pulse".PhtOver)
   END_RUNG wire#w2
   RUNG wire#w1
      P_Contact(operand := "ProcessAlarms".PhtReportDataNotLogged, bit := "pulse".PhtReportDataNotLogged)
   END_RUNG wire#w2
   RUNG wire#w1
      P_Contact(operand := "ProcessAlarms".SterilizationTimeOver, bit := "pulse".SterilizationTimeOver)
   END_RUNG wire#w2
   RUNG wire#w1
      P_Contact(operand := "ProcessAlarms".SteamFlowLow, bit := "pulse".SteamFlowLow)
   END_RUNG wire#w2
   RUNG wire#w1
      P_Contact(operand := "ProcessAlarms".SterilizationHighTemperature, bit := "pulse".SterilizationHighTemperature)
   END_RUNG wire#w2
   RUNG wire#w1
      P_Contact(operand := "ProcessAlarms".SterilizationCycleCompleted, bit := "pulse".SterilizationCycleCompleted)
   END_RUNG wire#w2
   RUNG wire#w1
      P_Contact(operand := "ProcessAlarms".SterilizationReportDataNotLogged, bit := "pulse".SterilizationReportDataNotLogged)
   END_RUNG wire#w2
   RUNG wire#w1
      P_Contact(operand := "ProcessAlarms".WfiFlowLow, bit := "pulse".WfiFlowLow)
   END_RUNG wire#w2
   RUNG wire#w1
      P_Contact(operand := "ProcessAlarms".BatchWfiFlowLow, bit := "pulse".BatchReportDataNotLogged)
   END_RUNG wire#w2
   // the same network as SCL:
   #_w1 := "AlwaysTRUE" AND "SafetyAlarms".ControlKeyOff AND NOT "pulse".ControlKeyOff;   // rising edge of "SafetyAlarms".ControlKeyOff
   "pulse".ControlKeyOff := "SafetyAlarms".ControlKeyOff;
   #_w2 := "AlwaysTRUE" AND "SafetyAlarms".EmergencyStopPressed AND NOT "pulse".EmergencyStopPressed;   // rising edge of "SafetyAlarms".EmergencyStopPressed
   "pulse".EmergencyStopPressed := "SafetyAlarms".EmergencyStopPressed;
   #_w3 := "AlwaysTRUE" AND "SafetyAlarms".PowerReset AND NOT "pulse".PowerReset;   // rising edge of "SafetyAlarms".PowerReset
   "pulse".PowerReset := "SafetyAlarms".PowerReset;
   #_w4 := "AlwaysTRUE" AND "SafetyAlarms".CompresseDairPressurelow AND NOT "pulse".CompresseDairPressurelow;   // rising edge of "SafetyAlarms".CompresseDairPressurelow
   "pulse".CompresseDairPressurelow := "SafetyAlarms".CompresseDairPressurelow;
   #_w5 := "AlwaysTRUE" AND "SafetyAlarms".PowerFailure AND NOT "pulse".PowerFailure;   // rising edge of "SafetyAlarms".PowerFailure
   "pulse".PowerFailure := "SafetyAlarms".PowerFailure;
   #_w6 := "AlwaysTRUE" AND "SafetyAlarms".PlcRestarted AND NOT "pulse".PlcRestarted;   // rising edge of "SafetyAlarms".PlcRestarted
   "pulse".PlcRestarted := "SafetyAlarms".PlcRestarted;
   #_w7 := "AlwaysTRUE" AND "SafetyAlarms".Mm01FeedbackTrip AND NOT "pulse".Mm01FeedbackTrip;   // rising edge of "SafetyAlarms".Mm01FeedbackTrip
   "pulse".Mm01FeedbackTrip := "SafetyAlarms".Mm01FeedbackTrip;
   #_w8 := "AlwaysTRUE" AND "SafetyAlarms".Cp01FeedbackTrip AND NOT "pulse".Cp01FeedbackTrip;   // rising edge of "SafetyAlarms".Cp01FeedbackTrip
   "pulse".Cp01FeedbackTrip := "SafetyAlarms".Cp01FeedbackTrip;
   #_w9 := "AlwaysTRUE" AND "SafetyAlarms".Mm01OverloadTrip AND NOT "pulse".Mm01OverloadTrip;   // rising edge of "SafetyAlarms".Mm01OverloadTrip
   "pulse".Mm01OverloadTrip := "SafetyAlarms".Mm01OverloadTrip;
   #_w10 := "AlwaysTRUE" AND "SafetyAlarms".Cp01OverloadTrip AND NOT "pulse".Cp01OverloadTrip;   // rising edge of "SafetyAlarms".Cp01OverloadTrip
   "pulse".Cp01OverloadTrip := "SafetyAlarms".Cp01OverloadTrip;
   #_w11 := "AlwaysTRUE" AND "SafetyAlarms".MinimumWeightRequiredToStartmm01 AND NOT "pulse".MinimumWeightRequiredToStartmm01;   // rising edge of "SafetyAlarms".MinimumWeightRequiredToStartmm01
   "pulse".MinimumWeightRequiredToStartmm01 := "SafetyAlarms".MinimumWeightRequiredToStartmm01;
   #_w12 := "AlwaysTRUE" AND "SafetyAlarms".Ticr01WireBreak AND NOT "pulse".Ticr01WireBreak;   // rising edge of "SafetyAlarms".Ticr01WireBreak
   "pulse".Ticr01WireBreak := "SafetyAlarms".Ticr01WireBreak;
   #_w13 := "AlwaysTRUE" AND "SafetyAlarms".Ticr02WireBreak AND NOT "pulse".Ticr02WireBreak;   // rising edge of "SafetyAlarms".Ticr02WireBreak
   "pulse".Ticr02WireBreak := "SafetyAlarms".Ticr02WireBreak;
   #_w14 := "AlwaysTRUE" AND "SafetyAlarms".Ticr03WireBreak AND NOT "pulse".Ticr03WireBreak;   // rising edge of "SafetyAlarms".Ticr03WireBreak
   "pulse".Ticr03WireBreak := "SafetyAlarms".Ticr03WireBreak;
   #_w15 := "AlwaysTRUE" AND "SafetyAlarms".Ticr04WireBreak AND NOT "pulse".Ticr04WireBreak;   // rising edge of "SafetyAlarms".Ticr04WireBreak
   "pulse".Ticr04WireBreak := "SafetyAlarms".Ticr04WireBreak;
   #_w16 := "AlwaysTRUE" AND "SafetyAlarms".Ticr05WireBreak AND NOT "pulse".Ticr05WireBreak;   // rising edge of "SafetyAlarms".Ticr05WireBreak
   "pulse".Ticr05WireBreak := "SafetyAlarms".Ticr05WireBreak;
   #_w17 := "AlwaysTRUE" AND "SafetyAlarms".Ticr06WireBreak AND NOT "pulse".Ticr06WireBreak;   // rising edge of "SafetyAlarms".Ticr06WireBreak
   "pulse".Ticr06WireBreak := "SafetyAlarms".Ticr06WireBreak;
   #_w18 := "AlwaysTRUE" AND "SafetyAlarms".Ticr07WireBreak AND NOT "pulse".Ticr07WireBreak;   // rising edge of "SafetyAlarms".Ticr07WireBreak
   "pulse".Ticr07WireBreak := "SafetyAlarms".Ticr07WireBreak;
   #_w19 := "AlwaysTRUE" AND "SafetyAlarms".Ticr08WireBreak AND NOT "pulse".Ticr08WireBreak;   // rising edge of "SafetyAlarms".Ticr08WireBreak
   "pulse".Ticr08WireBreak := "SafetyAlarms".Ticr08WireBreak;
   #_w20 := "AlwaysTRUE" AND "SafetyAlarms".Ticr09WireBreak AND NOT "pulse".Ticr09WireBreak;   // rising edge of "SafetyAlarms".Ticr09WireBreak
   "pulse".Ticr09WireBreak := "SafetyAlarms".Ticr09WireBreak;
   #_w21 := "AlwaysTRUE" AND "SafetyAlarms".Ticr10WireBreak AND NOT "pulse".Ticr10WireBreak;   // rising edge of "SafetyAlarms".Ticr10WireBreak
   "pulse".Ticr10WireBreak := "SafetyAlarms".Ticr10WireBreak;
   #_w22 := "AlwaysTRUE" AND "SafetyAlarms".Picr01WireBreak AND NOT "pulse".Picr01WireBreak;   // rising edge of "SafetyAlarms".Picr01WireBreak
   "pulse".Picr01WireBreak := "SafetyAlarms".Picr01WireBreak;
   #_w23 := "AlwaysTRUE" AND "SafetyAlarms".Picr02WireBreak AND NOT "pulse".Picr02WireBreak;   // rising edge of "SafetyAlarms".Picr02WireBreak
   "pulse".Picr02WireBreak := "SafetyAlarms".Picr02WireBreak;
   #_w24 := "AlwaysTRUE" AND "SafetyAlarms".Picr03WireBreak AND NOT "pulse".Picr03WireBreak;   // rising edge of "SafetyAlarms".Picr03WireBreak
   "pulse".Picr03WireBreak := "SafetyAlarms".Picr03WireBreak;
   #_w25 := "AlwaysTRUE" AND "SafetyAlarms".Picr04WireBreak AND NOT "pulse".Picr04WireBreak;   // rising edge of "SafetyAlarms".Picr04WireBreak
   "pulse".Picr04WireBreak := "SafetyAlarms".Picr04WireBreak;
   #_w26 := "AlwaysTRUE" AND "SafetyAlarms".Cicr01WireBreak AND NOT "pulse".Cicr01WireBreak;   // rising edge of "SafetyAlarms".Cicr01WireBreak
   "pulse".Cicr01WireBreak := "SafetyAlarms".Cicr01WireBreak;
   #_w27 := "AlwaysTRUE" AND "SafetyAlarms".Lc01CommunicationFailed AND NOT "pulse".Lc01CommunicationFailed;   // rising edge of "SafetyAlarms".Lc01CommunicationFailed
   "pulse".Lc01CommunicationFailed := "SafetyAlarms".Lc01CommunicationFailed;
   #_w28 := "AlwaysTRUE" AND "SafetyAlarms".VesselHighPressure AND NOT "pulse".VesselHighPressure;   // rising edge of "SafetyAlarms".VesselHighPressure
   "pulse".VesselHighPressure := "SafetyAlarms".VesselHighPressure;
   #_w29 := "AlwaysTRUE" AND "SafetyAlarms".Mm01SpeedSensorTrip AND NOT "pulse".Mm01SpeedSensorTrip;   // rising edge of "SafetyAlarms".Mm01SpeedSensorTrip
   "pulse".Mm01SpeedSensorTrip := "SafetyAlarms".Mm01SpeedSensorTrip;
   #_w30 := "AlwaysTRUE" AND "SafetyAlarms".PlcToHmiCommunicationFailed AND NOT "pulse".PlcToHmiCommunicationFailed;   // rising edge of "SafetyAlarms".PlcToHmiCommunicationFailed
   "pulse".PlcToHmiCommunicationFailed := "SafetyAlarms".PlcToHmiCommunicationFailed;
   #_w31 := "AlwaysTRUE" AND "ProcessAlarms".CipCycleOver AND NOT "pulse".CipCycleOver;   // rising edge of "ProcessAlarms".CipCycleOver
   "pulse".CipCycleOver := "ProcessAlarms".CipCycleOver;
   #_w32 := "AlwaysTRUE" AND "ProcessAlarms".CipCycleConductivityReached AND NOT "pulse".CipCycleConductivityReached;   // rising edge of "ProcessAlarms".CipCycleConductivityReached
   "pulse".CipCycleConductivityReached := "ProcessAlarms".CipCycleConductivityReached;
   #_w33 := "AlwaysTRUE" AND "ProcessAlarms".CipCycleConductivityNotReached AND NOT "pulse".CipCycleConductivityNotReached;   // rising edge of "ProcessAlarms".CipCycleConductivityNotReached
   "pulse".CipCycleConductivityNotReached := "ProcessAlarms".CipCycleConductivityNotReached;
   #_w34 := "AlwaysTRUE" AND "ProcessAlarms".ConductivityNotSampled AND NOT "pulse".ConductivityNotSampled;   // rising edge of "ProcessAlarms".ConductivityNotSampled
   "pulse".ConductivityNotSampled := "ProcessAlarms".ConductivityNotSampled;
   #_w35 := "AlwaysTRUE" AND "ProcessAlarms".CipReportDataNotLogged AND NOT "pulse".CipReportDataNotLogged;   // rising edge of "ProcessAlarms".CipReportDataNotLogged
   "pulse".CipReportDataNotLogged := "ProcessAlarms".CipReportDataNotLogged;
   #_w36 := "AlwaysTRUE" AND "ProcessAlarms".PhtFailed AND NOT "pulse".PhtFailed;   // rising edge of "ProcessAlarms".PhtFailed
   "pulse".PhtFailed := "ProcessAlarms".PhtFailed;
   #_w37 := "AlwaysTRUE" AND "ProcessAlarms".PhtPassed AND NOT "pulse".PhtPass;   // rising edge of "ProcessAlarms".PhtPassed
   "pulse".PhtPass := "ProcessAlarms".PhtPassed;
   #_w38 := "AlwaysTRUE" AND "ProcessAlarms".PhtOver AND NOT "pulse".PhtOver;   // rising edge of "ProcessAlarms".PhtOver
   "pulse".PhtOver := "ProcessAlarms".PhtOver;
   #_w39 := "AlwaysTRUE" AND "ProcessAlarms".PhtReportDataNotLogged AND NOT "pulse".PhtReportDataNotLogged;   // rising edge of "ProcessAlarms".PhtReportDataNotLogged
   "pulse".PhtReportDataNotLogged := "ProcessAlarms".PhtReportDataNotLogged;
   #_w40 := "AlwaysTRUE" AND "ProcessAlarms".SterilizationTimeOver AND NOT "pulse".SterilizationTimeOver;   // rising edge of "ProcessAlarms".SterilizationTimeOver
   "pulse".SterilizationTimeOver := "ProcessAlarms".SterilizationTimeOver;
   #_w41 := "AlwaysTRUE" AND "ProcessAlarms".SteamFlowLow AND NOT "pulse".SteamFlowLow;   // rising edge of "ProcessAlarms".SteamFlowLow
   "pulse".SteamFlowLow := "ProcessAlarms".SteamFlowLow;
   #_w42 := "AlwaysTRUE" AND "ProcessAlarms".SterilizationHighTemperature AND NOT "pulse".SterilizationHighTemperature;   // rising edge of "ProcessAlarms".SterilizationHighTemperature
   "pulse".SterilizationHighTemperature := "ProcessAlarms".SterilizationHighTemperature;
   #_w43 := "AlwaysTRUE" AND "ProcessAlarms".SterilizationCycleCompleted AND NOT "pulse".SterilizationCycleCompleted;   // rising edge of "ProcessAlarms".SterilizationCycleCompleted
   "pulse".SterilizationCycleCompleted := "ProcessAlarms".SterilizationCycleCompleted;
   #_w44 := "AlwaysTRUE" AND "ProcessAlarms".SterilizationReportDataNotLogged AND NOT "pulse".SterilizationReportDataNotLogged;   // rising edge of "ProcessAlarms".SterilizationReportDataNotLogged
   "pulse".SterilizationReportDataNotLogged := "ProcessAlarms".SterilizationReportDataNotLogged;
   #_w45 := "AlwaysTRUE" AND "ProcessAlarms".WfiFlowLow AND NOT "pulse".WfiFlowLow;   // rising edge of "ProcessAlarms".WfiFlowLow
   "pulse".WfiFlowLow := "ProcessAlarms".WfiFlowLow;
   #_w46 := "AlwaysTRUE" AND "ProcessAlarms".BatchWfiFlowLow AND NOT "pulse".BatchReportDataNotLogged;   // rising edge of "ProcessAlarms".BatchWfiFlowLow
   "pulse".BatchReportDataNotLogged := "ProcessAlarms".BatchWfiFlowLow;
   IF #_w1 OR #_w2 OR #_w3 OR #_w4 OR #_w5 OR #_w6 OR #_w7 OR #_w8 OR #_w9 OR #_w10 OR #_w11 OR #_w12 OR #_w13 OR #_w14 OR #_w15 OR #_w16 OR #_w17 OR #_w18 OR #_w19 OR #_w20 OR #_w21 OR #_w22 OR #_w23 OR #_w24 OR #_w25 OR #_w26 OR #_w27 OR #_w28 OR #_w29 OR #_w30 OR #_w31 OR #_w32 OR #_w33 OR #_w34 OR #_w35 OR #_w36 OR #_w37 OR #_w38 OR #_w39 OR #_w40 OR #_w41 OR #_w42 OR #_w43 OR #_w44 OR #_w45 OR #_w46 THEN
       "HmiTags".Hooter := TRUE;
   END_IF;
END_REGION

REGION Network 31: "HmiTags".Hooter -- reset
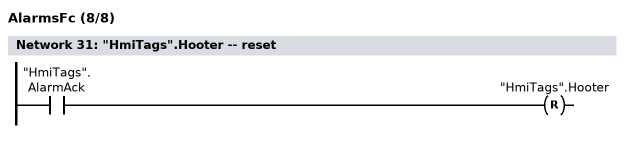
   RUNG wire#powerrail
      Contact( "HmiTags".AlarmAck )
      R_Coil( "HmiTags".Hooter )
   END_RUNG
   // the same network as SCL:
   IF "HmiTags".AlarmAck THEN "HmiTags".Hooter := FALSE; END_IF;
END_REGION
END_FUNCTION

FUNCTION "PHT_Logic" : Void   // FC1206, LAD
{ S7_Optimized_Access := 'FALSE' }
// stored: AutoNumber false, SetENOAutomatically false
   VAR_TEMP   // added for the SCL form of the ladder/FBD networks
      _w1 : Bool;
      _w2 : Bool;
      _w3 : Bool;
      _w4 : Bool;
      _w5 : Bool;
      _w6 : Bool;
      _w7 : Bool;
   END_VAR
BEGIN

REGION Network 1: "PHT Cycle".Start
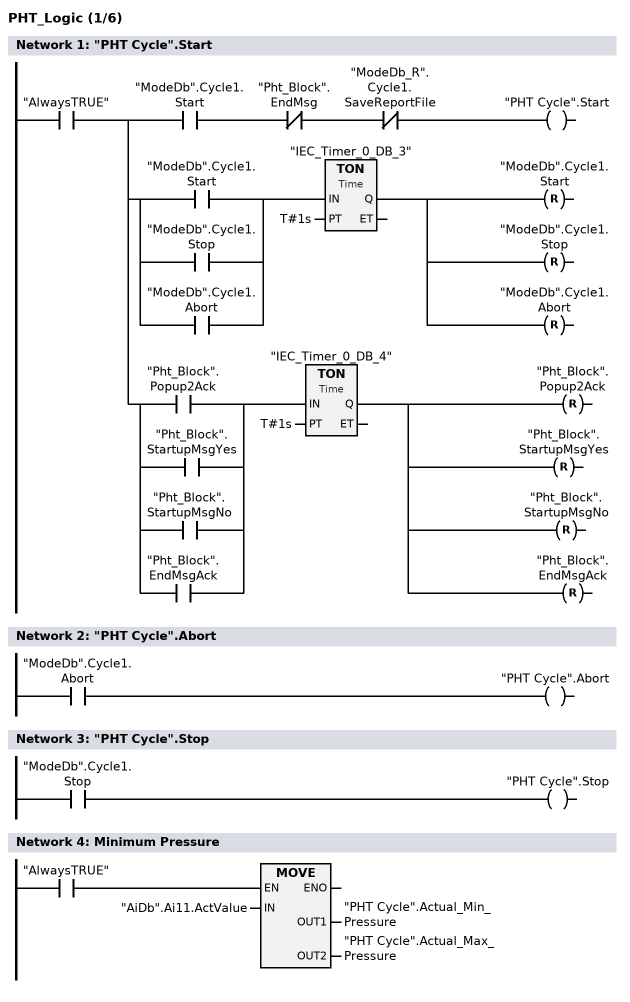
   RUNG wire#powerrail
      Contact( "AlwaysTRUE" )
      wire#w1
      Contact( "ModeDb".Cycle1.Start )
      I_Contact( "Pht_Block".EndMsg )
      I_Contact( "ModeDb_R".Cycle1.SaveReportFile )
      Coil( "PHT Cycle".Start )
   END_RUNG
   RUNG wire#w1
      Contact( "ModeDb".Cycle1.Start )
      wire#w2
      { S7_Templates := "time_type := Time" } "IEC_Timer_0_DB_3".TON(pt := T#1s, et =>)
      wire#w3
      R_Coil( "ModeDb".Cycle1.Start )
   END_RUNG
   RUNG wire#w1
      Contact( "ModeDb".Cycle1.Stop )
   END_RUNG wire#w2
   RUNG wire#w1
      Contact( "ModeDb".Cycle1.Abort )
   END_RUNG wire#w2
   RUNG wire#w3
      R_Coil( "ModeDb".Cycle1.Stop )
   END_RUNG
   RUNG wire#w3
      R_Coil( "ModeDb".Cycle1.Abort )
   END_RUNG
   RUNG wire#w1
      Contact( "Pht_Block".Popup2Ack )
      wire#w4
      { S7_Templates := "time_type := Time" } "IEC_Timer_0_DB_4".TON(pt := T#1s, et =>)
      wire#w5
      R_Coil( "Pht_Block".Popup2Ack )
   END_RUNG
   RUNG wire#w1
      Contact( "Pht_Block".StartupMsgYes )
   END_RUNG wire#w4
   RUNG wire#w1
      Contact( "Pht_Block".StartupMsgNo )
   END_RUNG wire#w4
   RUNG wire#w1
      Contact( "Pht_Block".EndMsgAck )
   END_RUNG wire#w4
   RUNG wire#w5
      R_Coil( "Pht_Block".StartupMsgYes )
   END_RUNG
   RUNG wire#w5
      R_Coil( "Pht_Block".StartupMsgNo )
   END_RUNG
   RUNG wire#w5
      R_Coil( "Pht_Block".EndMsgAck )
   END_RUNG
   // the same network as SCL:
   "PHT Cycle".Start := "AlwaysTRUE" AND "ModeDb".Cycle1.Start AND NOT "Pht_Block".EndMsg AND NOT "ModeDb_R".Cycle1.SaveReportFile;
   "IEC_Timer_0_DB_3".TON(IN := "AlwaysTRUE" AND ("ModeDb".Cycle1.Start OR "ModeDb".Cycle1.Stop OR "ModeDb".Cycle1.Abort),
                          PT := T#1s);
   IF "IEC_Timer_0_DB_3".Q THEN
       "ModeDb".Cycle1.Start := FALSE;
       "ModeDb".Cycle1.Stop := FALSE;
       "ModeDb".Cycle1.Abort := FALSE;
   END_IF;
   "IEC_Timer_0_DB_4".TON(IN := "AlwaysTRUE" AND ("Pht_Block".Popup2Ack OR "Pht_Block".StartupMsgYes OR "Pht_Block".StartupMsgNo OR "Pht_Block".EndMsgAck),
                          PT := T#1s);
   IF "IEC_Timer_0_DB_4".Q THEN
       "Pht_Block".Popup2Ack := FALSE;
       "Pht_Block".StartupMsgYes := FALSE;
       "Pht_Block".StartupMsgNo := FALSE;
       "Pht_Block".EndMsgAck := FALSE;
   END_IF;
END_REGION

REGION Network 2: "PHT Cycle".Abort
   RUNG wire#powerrail
      Contact( "ModeDb".Cycle1.Abort )
      Coil( "PHT Cycle".Abort )
   END_RUNG
   // the same network as SCL:
   "PHT Cycle".Abort := "ModeDb".Cycle1.Abort;
END_REGION

REGION Network 3: "PHT Cycle".Stop
   RUNG wire#powerrail
      Contact( "ModeDb".Cycle1.Stop )
      Coil( "PHT Cycle".Stop )
   END_RUNG
   // the same network as SCL:
   "PHT Cycle".Stop := "ModeDb".Cycle1.Stop;
END_REGION

REGION Network 4: Minimum Pressure
   RUNG wire#powerrail
      Contact( "AlwaysTRUE" )
      Move(in := "AiDb".Ai11.ActValue, out1 => "PHT Cycle".Actual_Min_Pressure, out2 => "PHT Cycle".Actual_Max_Pressure)
   END_RUNG
   // the same network as SCL:
   IF "AlwaysTRUE" THEN
       "PHT Cycle".Actual_Min_Pressure := "AiDb".Ai11.ActValue;
       "PHT Cycle".Actual_Max_Pressure := "AiDb".Ai11.ActValue;
   END_IF;
END_REGION

REGION Network 5: "PHT Cycle".fault
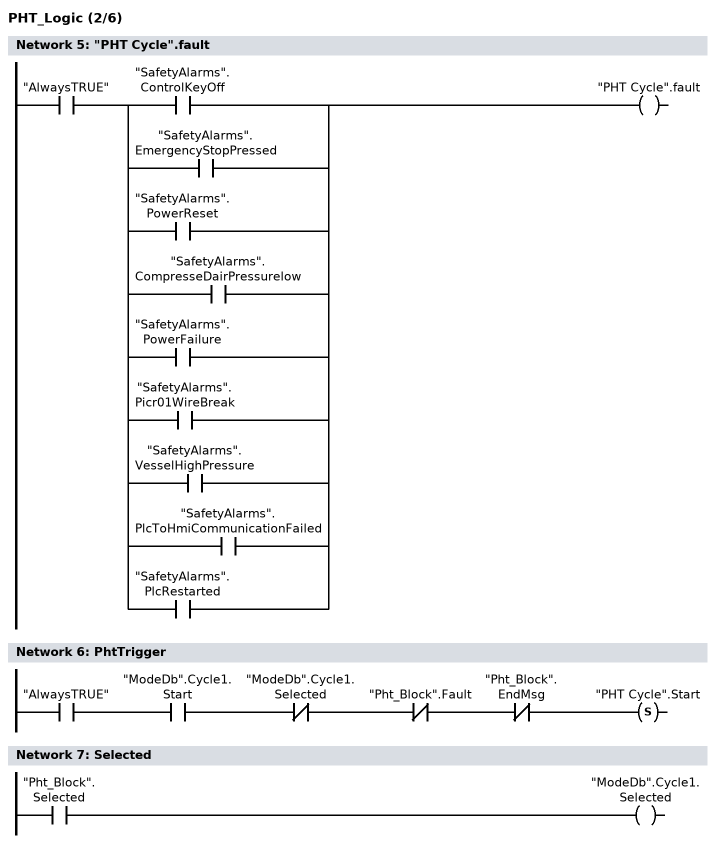
   RUNG wire#powerrail
      Contact( "AlwaysTRUE" )
      wire#w1
      Contact( "SafetyAlarms".ControlKeyOff )
      wire#w2
      Coil( "PHT Cycle".fault )
   END_RUNG
   RUNG wire#w1
      Contact( "SafetyAlarms".EmergencyStopPressed )
   END_RUNG wire#w2
   RUNG wire#w1
      Contact( "SafetyAlarms".PowerReset )
   END_RUNG wire#w2
   RUNG wire#w1
      Contact( "SafetyAlarms".CompresseDairPressurelow )
   END_RUNG wire#w2
   RUNG wire#w1
      Contact( "SafetyAlarms".PowerFailure )
   END_RUNG wire#w2
   RUNG wire#w1
      Contact( "SafetyAlarms".Picr01WireBreak )
   END_RUNG wire#w2
   RUNG wire#w1
      Contact( "SafetyAlarms".VesselHighPressure )
   END_RUNG wire#w2
   RUNG wire#w1
      Contact( "SafetyAlarms".PlcToHmiCommunicationFailed )
   END_RUNG wire#w2
   RUNG wire#w1
      Contact( "SafetyAlarms".PlcRestarted )
   END_RUNG wire#w2
   // the same network as SCL:
   "PHT Cycle".fault := "AlwaysTRUE" AND ("SafetyAlarms".ControlKeyOff OR "SafetyAlarms".EmergencyStopPressed OR "SafetyAlarms".PowerReset OR "SafetyAlarms".CompresseDairPressurelow OR "SafetyAlarms".PowerFailure OR "SafetyAlarms".Picr01WireBreak OR "SafetyAlarms".VesselHighPressure OR "SafetyAlarms".PlcToHmiCommunicationFailed OR "SafetyAlarms".PlcRestarted);
END_REGION

REGION Network 6: PhtTrigger
   RUNG wire#powerrail
      Contact( "AlwaysTRUE" )
      Contact( "ModeDb".Cycle1.Start )
      I_Contact( "ModeDb".Cycle1.Selected )
      I_Contact( "Pht_Block".Fault )
      I_Contact( "Pht_Block".EndMsg )
      S_Coil( "PHT Cycle".Start )
   END_RUNG
   // the same network as SCL:
   IF "AlwaysTRUE" AND "ModeDb".Cycle1.Start AND NOT "ModeDb".Cycle1.Selected AND NOT "Pht_Block".Fault AND NOT "Pht_Block".EndMsg THEN
       "PHT Cycle".Start := TRUE;
   END_IF;
END_REGION

REGION Network 7: Selected
   RUNG wire#powerrail
      Contact( "Pht_Block".Selected )
      Coil( "ModeDb".Cycle1.Selected )
   END_RUNG
   // the same network as SCL:
   "ModeDb".Cycle1.Selected := "Pht_Block".Selected;
END_REGION

REGION Network 8: PHT Block
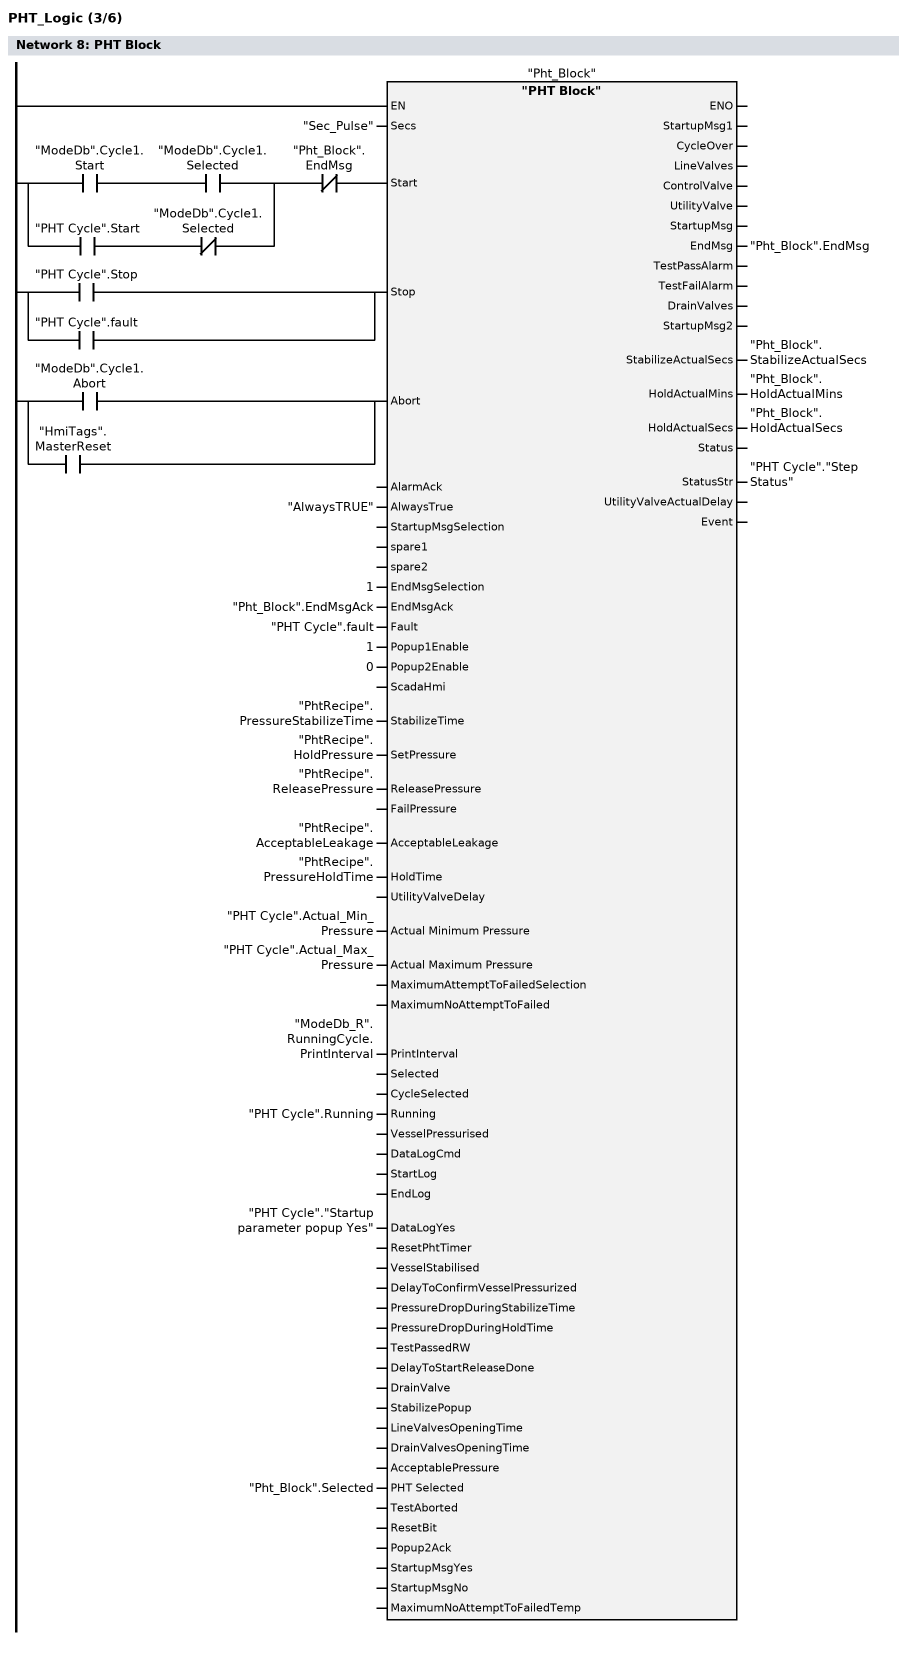
   RUNG wire#powerrail
      "Pht_Block"(Start := wire#w2, Stop := wire#w3, Abort := wire#w4, Secs := "Sec_Pulse", AlarmAck :=, AlwaysTrue := "AlwaysTRUE", StartupMsgSelection :=, spare1 :=, spare2 :=, EndMsgSelection := 1, EndMsgAck := "Pht_Block".EndMsgAck, Fault := "PHT Cycle".fault, Popup1Enable := 1, Popup2Enable := 0, ScadaHmi :=, StabilizeTime := "PhtRecipe".PressureStabilizeTime, SetPressure := "PhtRecipe".HoldPressure, ReleasePressure := "PhtRecipe".ReleasePressure, FailPressure :=, AcceptableLeakage := "PhtRecipe".AcceptableLeakage, HoldTime := "PhtRecipe".PressureHoldTime, UtilityValveDelay :=, "Actual Minimum Pressure" := "PHT Cycle".Actual_Min_Pressure, "Actual Maximum Pressure" := "PHT Cycle".Actual_Max_Pressure, MaximumAttemptToFailedSelection :=, MaximumNoAttemptToFailed :=, PrintInterval := "ModeDb_R".RunningCycle.PrintInterval, Selected :=, CycleSelected :=, Running := "PHT Cycle".Running, VesselPressurised :=, DataLogCmd :=, StartLog :=, EndLog :=, DataLogYes := "PHT Cycle"."Startup parameter popup Yes", ResetPhtTimer :=, VesselStabilised :=, DelayToConfirmVesselPressurized :=, PressureDropDuringStabilizeTime :=, PressureDropDuringHoldTime :=, TestPassedRW :=, DelayToStartReleaseDone :=, DrainValve :=, StabilizePopup :=, LineValvesOpeningTime :=, DrainValvesOpeningTime :=, AcceptablePressure :=, "PHT Selected" := "Pht_Block".Selected, TestAborted :=, ResetBit :=, Popup2Ack :=, StartupMsgYes :=, StartupMsgNo :=, MaximumNoAttemptToFailedTemp :=, StartupMsg1 =>, CycleOver =>, LineValves =>, ControlValve =>, UtilityValve =>, StartupMsg =>, EndMsg => "Pht_Block".EndMsg, TestPassAlarm =>, TestFailAlarm =>, DrainValves =>, StartupMsg2 =>, StabilizeActualSecs => "Pht_Block".StabilizeActualSecs, HoldActualMins => "Pht_Block".HoldActualMins, HoldActualSecs => "Pht_Block".HoldActualSecs, Status =>, StatusStr => "PHT Cycle"."Step Status", UtilityValveActualDelay =>, Event =>)
   END_RUNG
   RUNG wire#powerrail
      Contact( "ModeDb".Cycle1.Start )
      Contact( "ModeDb".Cycle1.Selected )
      wire#w1
      I_Contact( "Pht_Block".EndMsg )
   END_RUNG wire#w2
   RUNG wire#powerrail
      Contact( "PHT Cycle".Start )
      I_Contact( "ModeDb".Cycle1.Selected )
   END_RUNG wire#w1
   RUNG wire#powerrail
      Contact( "PHT Cycle".Stop )
   END_RUNG wire#w3
   RUNG wire#powerrail
      Contact( "PHT Cycle".fault )
   END_RUNG wire#w3
   RUNG wire#powerrail
      Contact( "ModeDb".Cycle1.Abort )
   END_RUNG wire#w4
   RUNG wire#powerrail
      Contact( "HmiTags".MasterReset )
   END_RUNG wire#w4
   // the same network as SCL:
   "Pht_Block"(Secs := "Sec_Pulse",   // "PHT Block"
               Start := (("ModeDb".Cycle1.Start AND "ModeDb".Cycle1.Selected) OR ("PHT Cycle".Start AND NOT "ModeDb".Cycle1.Selected)) AND NOT "Pht_Block".EndMsg,
               Stop := "PHT Cycle".Stop OR "PHT Cycle".fault,
               Abort := "ModeDb".Cycle1.Abort OR "HmiTags".MasterReset,
               AlwaysTrue := "AlwaysTRUE",
               EndMsgSelection := 1,
               EndMsgAck := "Pht_Block".EndMsgAck,
               Fault := "PHT Cycle".fault,
               Popup1Enable := 1,
               Popup2Enable := 0,
               StabilizeTime := "PhtRecipe".PressureStabilizeTime,
               SetPressure := "PhtRecipe".HoldPressure,
               ReleasePressure := "PhtRecipe".ReleasePressure,
               AcceptableLeakage := "PhtRecipe".AcceptableLeakage,
               HoldTime := "PhtRecipe".PressureHoldTime,
               "Actual Minimum Pressure" := "PHT Cycle".Actual_Min_Pressure,
               "Actual Maximum Pressure" := "PHT Cycle".Actual_Max_Pressure,
               PrintInterval := "ModeDb_R".RunningCycle.PrintInterval,
               Running := "PHT Cycle".Running,
               DataLogYes := "PHT Cycle"."Startup parameter popup Yes",
               "PHT Selected" := "Pht_Block".Selected,
               EndMsg => "Pht_Block".EndMsg,
               StabilizeActualSecs => "Pht_Block".StabilizeActualSecs,
               HoldActualMins => "Pht_Block".HoldActualMins,
               HoldActualSecs => "Pht_Block".HoldActualSecs,
               StatusStr => "PHT Cycle"."Step Status");
END_REGION

REGION Network 9: PHT ALARMS
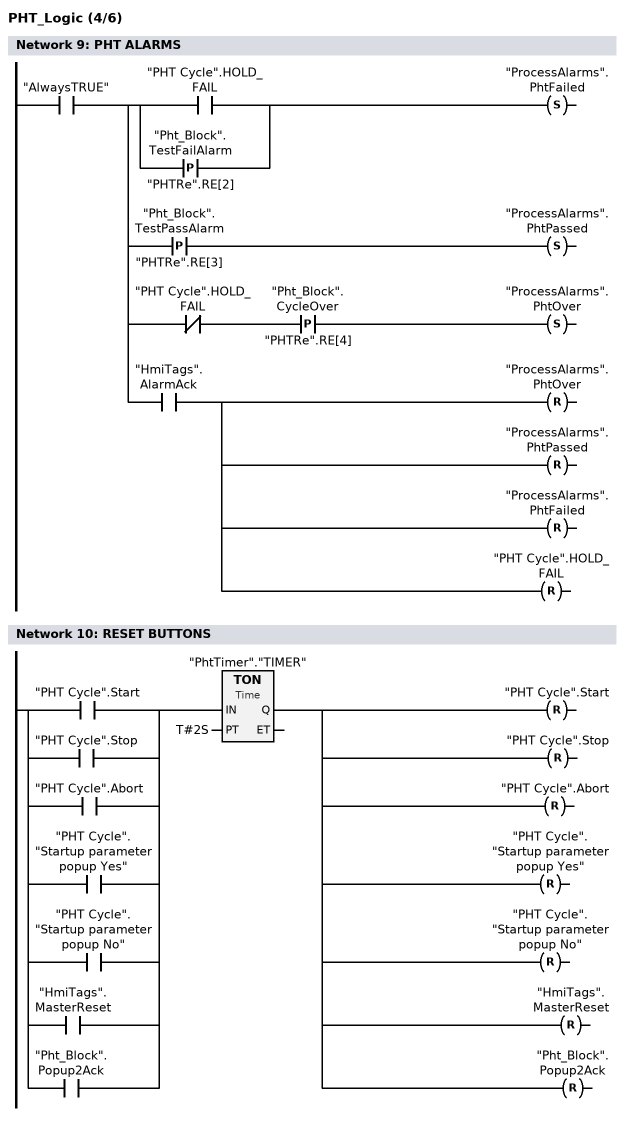
   RUNG wire#powerrail
      Contact( "AlwaysTRUE" )
      wire#w1
      Contact( "PHT Cycle".HOLD_FAIL )
      wire#w2
      S_Coil( "ProcessAlarms".PhtFailed )
   END_RUNG
   RUNG wire#w1
      P_Contact(operand := "Pht_Block".TestFailAlarm, bit := "PHTRe".RE[2])
   END_RUNG wire#w2
   RUNG wire#w1
      P_Contact(operand := "Pht_Block".TestPassAlarm, bit := "PHTRe".RE[3])
      S_Coil( "ProcessAlarms".PhtPassed )
   END_RUNG
   RUNG wire#w1
      I_Contact( "PHT Cycle".HOLD_FAIL )
      P_Contact(operand := "Pht_Block".CycleOver, bit := "PHTRe".RE[4])
      S_Coil( "ProcessAlarms".PhtOver )
   END_RUNG
   RUNG wire#w1
      Contact( "HmiTags".AlarmAck )
      wire#w3
      R_Coil( "ProcessAlarms".PhtOver )
   END_RUNG
   RUNG wire#w3
      R_Coil( "ProcessAlarms".PhtPassed )
   END_RUNG
   RUNG wire#w3
      R_Coil( "ProcessAlarms".PhtFailed )
   END_RUNG
   RUNG wire#w3
      R_Coil( "PHT Cycle".HOLD_FAIL )
   END_RUNG
   // the same network as SCL:
   #_w1 := "AlwaysTRUE" AND "Pht_Block".TestFailAlarm AND NOT "PHTRe".RE[2];   // rising edge of "Pht_Block".TestFailAlarm
   "PHTRe".RE[2] := "Pht_Block".TestFailAlarm;
   IF ("AlwaysTRUE" AND "PHT Cycle".HOLD_FAIL) OR #_w1 THEN "ProcessAlarms".PhtFailed := TRUE; END_IF;
   #_w2 := "AlwaysTRUE" AND "Pht_Block".TestPassAlarm AND NOT "PHTRe".RE[3];   // rising edge of "Pht_Block".TestPassAlarm
   "PHTRe".RE[3] := "Pht_Block".TestPassAlarm;
   IF #_w2 THEN "ProcessAlarms".PhtPassed := TRUE; END_IF;
   #_w3 := "AlwaysTRUE" AND NOT "PHT Cycle".HOLD_FAIL AND "Pht_Block".CycleOver AND NOT "PHTRe".RE[4];   // rising edge of "Pht_Block".CycleOver
   "PHTRe".RE[4] := "Pht_Block".CycleOver;
   IF #_w3 THEN "ProcessAlarms".PhtOver := TRUE; END_IF;
   IF "AlwaysTRUE" AND "HmiTags".AlarmAck THEN
       "ProcessAlarms".PhtOver := FALSE;
       "ProcessAlarms".PhtPassed := FALSE;
       "ProcessAlarms".PhtFailed := FALSE;
       "PHT Cycle".HOLD_FAIL := FALSE;
   END_IF;
END_REGION

REGION Network 10: RESET BUTTONS
   RUNG wire#powerrail
      Contact( "PHT Cycle".Start )
      wire#w1
      { S7_Templates := "time_type := Time" } "PhtTimer"."TIMER".TON(pt := T#2S, et =>)
      wire#w2
      R_Coil( "PHT Cycle".Start )
   END_RUNG
   RUNG wire#powerrail
      Contact( "PHT Cycle".Stop )
   END_RUNG wire#w1
   RUNG wire#powerrail
      Contact( "PHT Cycle".Abort )
   END_RUNG wire#w1
   RUNG wire#powerrail
      Contact( "PHT Cycle"."Startup parameter popup Yes" )
   END_RUNG wire#w1
   RUNG wire#powerrail
      Contact( "PHT Cycle"."Startup parameter popup No" )
   END_RUNG wire#w1
   RUNG wire#powerrail
      Contact( "HmiTags".MasterReset )
   END_RUNG wire#w1
   RUNG wire#powerrail
      Contact( "Pht_Block".Popup2Ack )
   END_RUNG wire#w1
   RUNG wire#w2
      R_Coil( "PHT Cycle".Stop )
   END_RUNG
   RUNG wire#w2
      R_Coil( "PHT Cycle".Abort )
   END_RUNG
   RUNG wire#w2
      R_Coil( "PHT Cycle"."Startup parameter popup Yes" )
   END_RUNG
   RUNG wire#w2
      R_Coil( "PHT Cycle"."Startup parameter popup No" )
   END_RUNG
   RUNG wire#w2
      R_Coil( "HmiTags".MasterReset )
   END_RUNG
   RUNG wire#w2
      R_Coil( "Pht_Block".Popup2Ack )
   END_RUNG
   // the same network as SCL:
   "PhtTimer"."TIMER".TON(IN := "PHT Cycle".Start OR "PHT Cycle".Stop OR "PHT Cycle".Abort OR "PHT Cycle"."Startup parameter popup Yes" OR "PHT Cycle"."Startup parameter popup No" OR "HmiTags".MasterReset OR "Pht_Block".Popup2Ack,
                          PT := T#2S);
   IF "PhtTimer"."TIMER".Q THEN
       "PHT Cycle".Start := FALSE;
       "PHT Cycle".Stop := FALSE;
       "PHT Cycle".Abort := FALSE;
       "PHT Cycle"."Startup parameter popup Yes" := FALSE;
       "PHT Cycle"."Startup parameter popup No" := FALSE;
       "HmiTags".MasterReset := FALSE;
       "Pht_Block".Popup2Ack := FALSE;
   END_IF;
END_REGION

REGION Network 11: RESULT
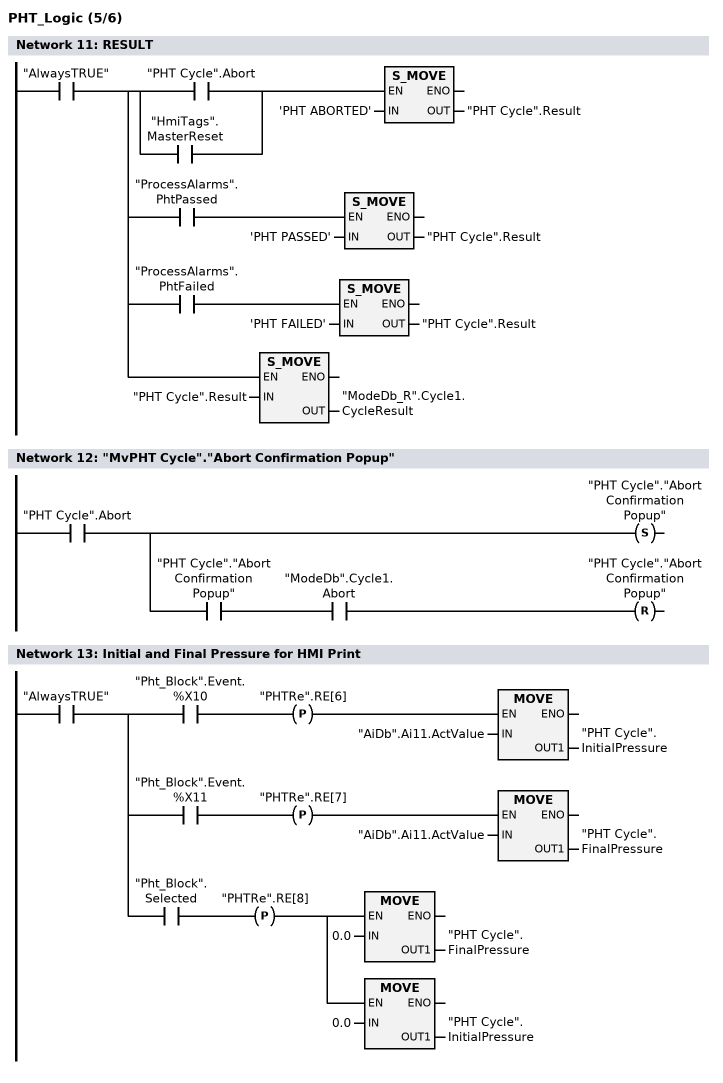
   RUNG wire#powerrail
      Contact( "AlwaysTRUE" )
      wire#w1
      Contact( "PHT Cycle".Abort )
      wire#w2
      S_Move(in := 'PHT ABORTED', out => "PHT Cycle".Result)
   END_RUNG
   RUNG wire#w1
      Contact( "HmiTags".MasterReset )
   END_RUNG wire#w2
   RUNG wire#w1
      Contact( "ProcessAlarms".PhtPassed )
      S_Move(in := 'PHT PASSED', out => "PHT Cycle".Result)
   END_RUNG
   RUNG wire#w1
      Contact( "ProcessAlarms".PhtFailed )
      S_Move(in := 'PHT FAILED', out => "PHT Cycle".Result)
   END_RUNG
   RUNG wire#w1
      S_Move(in := "PHT Cycle".Result, out => "ModeDb_R".Cycle1.CycleResult)
   END_RUNG
   // the same network as SCL:
   IF "AlwaysTRUE" AND ("PHT Cycle".Abort OR "HmiTags".MasterReset) THEN
       "PHT Cycle".Result := 'PHT ABORTED';
   END_IF;
   IF "AlwaysTRUE" AND "ProcessAlarms".PhtPassed THEN "PHT Cycle".Result := 'PHT PASSED'; END_IF;
   IF "AlwaysTRUE" AND "ProcessAlarms".PhtFailed THEN "PHT Cycle".Result := 'PHT FAILED'; END_IF;
   IF "AlwaysTRUE" THEN "ModeDb_R".Cycle1.CycleResult := "PHT Cycle".Result; END_IF;
END_REGION

REGION Network 12: "MvPHT Cycle"."Abort Confirmation Popup"
   RUNG wire#powerrail
      Contact( "PHT Cycle".Abort )
      wire#w1
      S_Coil( "PHT Cycle"."Abort Confirmation Popup" )
   END_RUNG
   RUNG wire#w1
      Contact( "PHT Cycle"."Abort Confirmation Popup" )
      Contact( "ModeDb".Cycle1.Abort )
      R_Coil( "PHT Cycle"."Abort Confirmation Popup" )
   END_RUNG
   // the same network as SCL:
   IF "PHT Cycle".Abort THEN "PHT Cycle"."Abort Confirmation Popup" := TRUE; END_IF;
   IF "PHT Cycle".Abort AND "PHT Cycle"."Abort Confirmation Popup" AND "ModeDb".Cycle1.Abort THEN
       "PHT Cycle"."Abort Confirmation Popup" := FALSE;
   END_IF;
END_REGION

REGION Network 13: Initial and Final Pressure for HMI Print
   RUNG wire#powerrail
      Contact( "AlwaysTRUE" )
      wire#w1
      Contact( "Pht_Block".Event.%X10 )
      P_Trig( "PHTRe".RE[6] )
      Move(in := "AiDb".Ai11.ActValue, out1 => "PHT Cycle".InitialPressure)
   END_RUNG
   RUNG wire#w1
      Contact( "Pht_Block".Event.%X11 )
      P_Trig( "PHTRe".RE[7] )
      Move(in := "AiDb".Ai11.ActValue, out1 => "PHT Cycle".FinalPressure)
   END_RUNG
   RUNG wire#w1
      Contact( "Pht_Block".Selected )
      P_Trig( "PHTRe".RE[8] )
      wire#w2
      Move(in := 0.0, out1 => "PHT Cycle".FinalPressure)
   END_RUNG
   RUNG wire#w2
      Move(in := 0.0, out1 => "PHT Cycle".InitialPressure)
   END_RUNG
   // the same network as SCL:
   #_w1 := "AlwaysTRUE" AND "Pht_Block".Event.%X10;
   #_w2 := #_w1 AND NOT "PHTRe".RE[6];   // rising edge
   "PHTRe".RE[6] := #_w1;
   IF #_w2 THEN "PHT Cycle".InitialPressure := "AiDb".Ai11.ActValue; END_IF;
   #_w3 := "AlwaysTRUE" AND "Pht_Block".Event.%X11;
   #_w4 := #_w3 AND NOT "PHTRe".RE[7];   // rising edge
   "PHTRe".RE[7] := #_w3;
   IF #_w4 THEN "PHT Cycle".FinalPressure := "AiDb".Ai11.ActValue; END_IF;
   #_w5 := "AlwaysTRUE" AND "Pht_Block".Selected;
   #_w6 := #_w5 AND NOT "PHTRe".RE[8];   // rising edge
   "PHTRe".RE[8] := #_w5;
   IF #_w6 THEN
       "PHT Cycle".FinalPressure := 0.0;
       "PHT Cycle".InitialPressure := 0.0;
   END_IF;
END_REGION

REGION Network 14: "PHT Cycle".HoldStartTimeLog
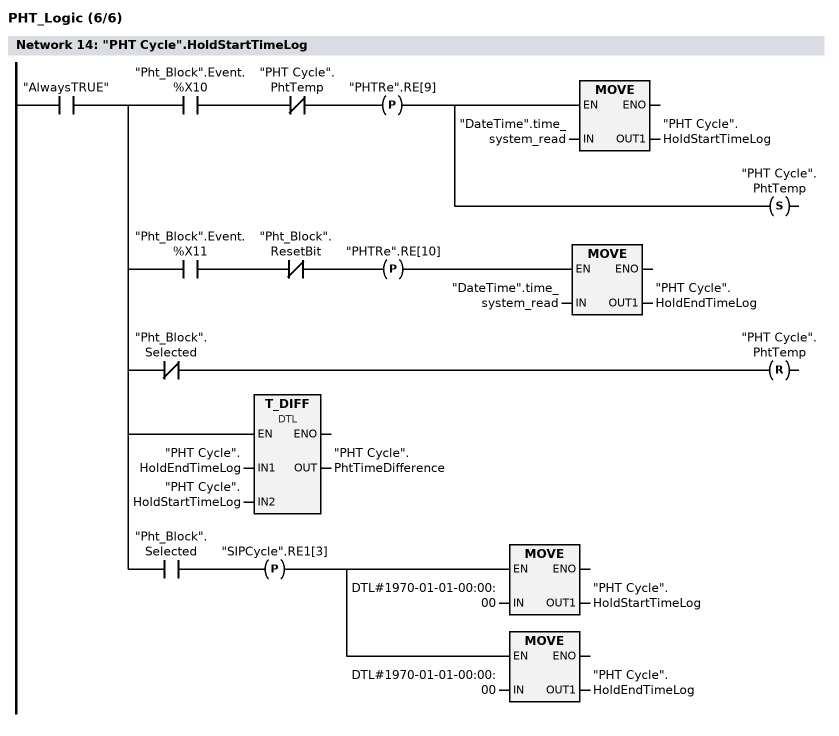
   RUNG wire#powerrail
      Contact( "AlwaysTRUE" )
      wire#w1
      Contact( "Pht_Block".Event.%X10 )
      I_Contact( "PHT Cycle".PhtTemp )
      P_Trig( "PHTRe".RE[9] )
      wire#w2
      Move(in := "DateTime".time_system_read, out1 => "PHT Cycle".HoldStartTimeLog)
   END_RUNG
   RUNG wire#w2
      S_Coil( "PHT Cycle".PhtTemp )
   END_RUNG
   RUNG wire#w1
      Contact( "Pht_Block".Event.%X11 )
      I_Contact( "Pht_Block".ResetBit )
      P_Trig( "PHTRe".RE[10] )
      Move(in := "DateTime".time_system_read, out1 => "PHT Cycle".HoldEndTimeLog)
   END_RUNG
   RUNG wire#w1
      I_Contact( "Pht_Block".Selected )
      R_Coil( "PHT Cycle".PhtTemp )
   END_RUNG
   RUNG wire#w1
      { S7_Templates := "[date_type := DTL, time_type := Time]" } T_DIFF(IN1 := "PHT Cycle".HoldEndTimeLog, IN2 := "PHT Cycle".HoldStartTimeLog, OUT => "PHT Cycle".PhtTimeDifference)
   END_RUNG
   RUNG wire#w1
      Contact( "Pht_Block".Selected )
      P_Trig( "SIPCycle".RE1[3] )
      wire#w3
      Move(in := DTL#1970-01-01-00:00:00, out1 => "PHT Cycle".HoldStartTimeLog)
   END_RUNG
   RUNG wire#w3
      Move(in := DTL#1970-01-01-00:00:00, out1 => "PHT Cycle".HoldEndTimeLog)
   END_RUNG
   // the same network as SCL:
   #_w1 := "AlwaysTRUE" AND "Pht_Block".Event.%X10 AND NOT "PHT Cycle".PhtTemp;
   #_w2 := #_w1 AND NOT "PHTRe".RE[9];   // rising edge
   "PHTRe".RE[9] := #_w1;
   IF #_w2 THEN
       "PHT Cycle".HoldStartTimeLog := "DateTime".time_system_read;
       "PHT Cycle".PhtTemp := TRUE;
   END_IF;
   #_w3 := "AlwaysTRUE" AND "Pht_Block".Event.%X11 AND NOT "Pht_Block".ResetBit;
   #_w4 := #_w3 AND NOT "PHTRe".RE[10];   // rising edge
   "PHTRe".RE[10] := #_w3;
   IF #_w4 THEN "PHT Cycle".HoldEndTimeLog := "DateTime".time_system_read; END_IF;
   IF "AlwaysTRUE" AND NOT "Pht_Block".Selected THEN "PHT Cycle".PhtTemp := FALSE; END_IF;
   #_w5 := "AlwaysTRUE";
   IF #_w5 THEN
       T_DIFF(IN1 := "PHT Cycle".HoldEndTimeLog,
              IN2 := "PHT Cycle".HoldStartTimeLog,
              OUT => "PHT Cycle".PhtTimeDifference);
   END_IF;
   #_w6 := #_w5 AND "Pht_Block".Selected;
   #_w7 := #_w6 AND NOT "SIPCycle".RE1[3];   // rising edge
   "SIPCycle".RE1[3] := #_w6;
   IF #_w7 THEN
       "PHT Cycle".HoldStartTimeLog := DTL#1970-01-01-00:00:00;
       "PHT Cycle".HoldEndTimeLog := DTL#1970-01-01-00:00:00;
   END_IF;
END_REGION

REGION Network 15 (SCL): SCL ROUNDOFF
   // Step 1: get TIME
   "PHT Cycle".TempTime := "PHT Cycle".PhtTimeDifference;

   // Step 2: TIME → milliseconds
   "PHT Cycle".TempMs := TIME_TO_DINT("PHT Cycle".TempTime);

   // Step 3: make positive (optional)
   //"PHT Cycle".TempMs := ABS("PHT Cycle".TempMs);

   // Step 4: ROUND milliseconds to seconds
   "PHT Cycle".TotalSecondsTag := ("PHT Cycle".TempMs + 500) / 1000;

   // Step 5: split HH MM SS
   "PHT Cycle".Hours := DINT_TO_INT("PHT Cycle".TotalSecondsTag / 3600);

   "PHT Cycle".Minutes := DINT_TO_INT(
   ("PHT Cycle".TotalSecondsTag MOD 3600) / 60
   );

   "PHT Cycle".Seconds := DINT_TO_INT(
    "PHT Cycle".TotalSecondsTag MOD 60
   );
END_REGION
END_FUNCTION

FUNCTION_BLOCK "PHT Block"   // FB401, LAD
{ S7_Optimized_Access := 'FALSE' }
// stored: AutoNumber false, SetENOAutomatically false
   VAR_INPUT
      Secs : Bool;
      Start : Bool;
      Stop : Bool;
      Abort : Bool;
      AlarmAck : Bool;
      AlwaysTrue : Bool;
      StartupMsgSelection : Bool;
      spare1 : Bool;
      spare2 : Bool;
      EndMsgSelection : Bool;
      EndMsgAck : Bool;
      Fault : Bool;
      Popup1Enable : Bool;
      Popup2Enable : Bool;
      ScadaHmi : Bool := 1;   // 0- scada, 1 - hmi
      StabilizeTime : Int;
      SetPressure : Real;
      ReleasePressure : Real;
      FailPressure : Real;
      AcceptableLeakage : Real;
      HoldTime : Int;
      UtilityValveDelay : Int;
      "Actual Minimum Pressure" : Real;
      "Actual Maximum Pressure" : Real;
      MaximumAttemptToFailedSelection : Int;
      MaximumNoAttemptToFailed : Int;
      PrintInterval : Int;
   END_VAR
   VAR_OUTPUT
      StartupMsg1 : Bool;
      CycleOver : Bool;
      LineValves : Bool;
      ControlValve : Bool;
      UtilityValve : Bool;
      StartupMsg : Bool;
      EndMsg : Bool;
      TestPassAlarm : Bool;
      TestFailAlarm : Bool;
      DrainValves : Bool;
      StartupMsg2 : Bool;
      StabilizeActualSecs : DInt;
      HoldActualMins : DInt;
      HoldActualSecs : DInt;
      Status : Int;
      StatusStr : String[60];
      UtilityValveActualDelay : Int;
      Event : Word;
   END_VAR
   VAR_IN_OUT
      Selected : Bool;
      CycleSelected : Bool;
      Running : Bool;
      VesselPressurised : Bool;
      DataLogCmd : Bool;
      StartLog : Bool;
      EndLog : Bool;
      DataLogYes : Bool;
      ResetPhtTimer : Bool;
      VesselStabilised : Bool;
      DelayToConfirmVesselPressurized : Bool;
      PressureDropDuringStabilizeTime : Bool;
      PressureDropDuringHoldTime : Bool;
      TestPassedRW : Bool;
      DelayToStartReleaseDone : Bool;
      DrainValve : Bool;
      StabilizePopup : Bool;
      LineValvesOpeningTime : Int;
      DrainValvesOpeningTime : Int;
      AcceptablePressure : Real;
      "PHT Selected" : Bool;
      TestAborted : Bool;
      ResetBit : Bool;
      Popup2Ack : Bool;
      StartupMsgYes : Bool;
      StartupMsgNo : Bool;
      MaximumNoAttemptToFailedTemp : Int;
   END_VAR
   VAR
      StabilizeTimer { S7_SetPoint := 'True'} : "R_TIMER";
      HoldTimer { S7_SetPoint := 'True'} : "R_TIMER";
      CheckPressureDuringStabilizeTime { S7_SetPoint := 'True'} : "On Delay Timer";
      CheckPressureDuringHoldTime { S7_SetPoint := 'True'} : "On Delay Timer";
      ReleaseCheckTime { S7_SetPoint := 'True'} : "On Delay Timer";
      CheckPressuredelay { S7_SetPoint := 'True'} : "On Delay Timer";
      DelayToStartRelease { S7_SetPoint := 'True'} : "On Delay Timer";
      StabilizeDelay { S7_SetPoint := 'True'} : "On Delay Timer";
      IEC_Timer_0_Instance { S7_SetPoint := 'True'} : TON_TIME;
      IEC_Timer_1_Instance { S7_SetPoint := 'True'} : TON_TIME;
      Timer1 { S7_SetPoint := 'True'} : TON_TIME;
      Timer2 { S7_SetPoint := 'True'} : TON_TIME;
      Timer3 { S7_SetPoint := 'True'} : TON_TIME;
      Timer4 { S7_SetPoint := 'True'} : TON_TIME;
      Timer5 { S7_SetPoint := 'True'} : TON_TIME;
      Timer6 { S7_SetPoint := 'True'} : TON_TIME;
      Timer7 { S7_SetPoint := 'True'} : TON_TIME;
      Re { ExternalAccessible := 'False'; ExternalVisible := 'False'; ExternalWritable := 'False'} : Bool;
      Re1 { ExternalAccessible := 'False'; ExternalVisible := 'False'; ExternalWritable := 'False'} : Bool;
      Re2 { ExternalAccessible := 'False'; ExternalVisible := 'False'; ExternalWritable := 'False'} : Bool;
      Re3 { ExternalAccessible := 'False'; ExternalVisible := 'False'; ExternalWritable := 'False'} : Bool;
      Re4 { ExternalAccessible := 'False'; ExternalVisible := 'False'; ExternalWritable := 'False'} : Bool;
      Re5 { ExternalAccessible := 'False'; ExternalVisible := 'False'; ExternalWritable := 'False'} : Bool;
      Re6 { ExternalAccessible := 'False'; ExternalVisible := 'False'; ExternalWritable := 'False'} : Bool;
      Re7 { ExternalAccessible := 'False'; ExternalVisible := 'False'; ExternalWritable := 'False'} : Bool;
      Re8 { ExternalAccessible := 'False'; ExternalVisible := 'False'; ExternalWritable := 'False'} : Bool;
      Re9 { ExternalAccessible := 'False'; ExternalVisible := 'False'; ExternalWritable := 'False'} : Bool;
      Re10 : Bool;
      Re11 : Bool;
      Re12 : Bool;
      Timer8 : TON_TIME;
      Timer9 { S7_SetPoint := 'True'} : TON_TIME;
      Timer10 { S7_SetPoint := 'True'} : TON_TIME;
      Timer11 { S7_SetPoint := 'True'} : TON_TIME;
      Timer12 { S7_SetPoint := 'True'} : TON_TIME;
      IEC_Counter_0_Instance { S7_SetPoint := 'True'} : CTU_INT;
      Re13 : Bool;
      Re14 : Bool;
      Re15 : Bool;
      timer13 : TON_TIME;
   END_VAR
   VAR_TEMP   // added for the SCL form of the ladder/FBD networks
      _w1 : Bool;
      _w2 : Bool;
      _w3 : Bool;
      _w4 : Bool;
      _w5 : Bool;
      _w6 : Bool;
      _w7 : Bool;
      _w8 : Bool;
      _w9 : Bool;
      _w10 : Bool;
      _w11 : Bool;
      _w12 : Bool;
      _w13 : Bool;
      _w14 : Bool;
      _w15 : Bool;
      _w16 : Bool;
   END_VAR
BEGIN

REGION Network 1: StartupMsgYesEnable
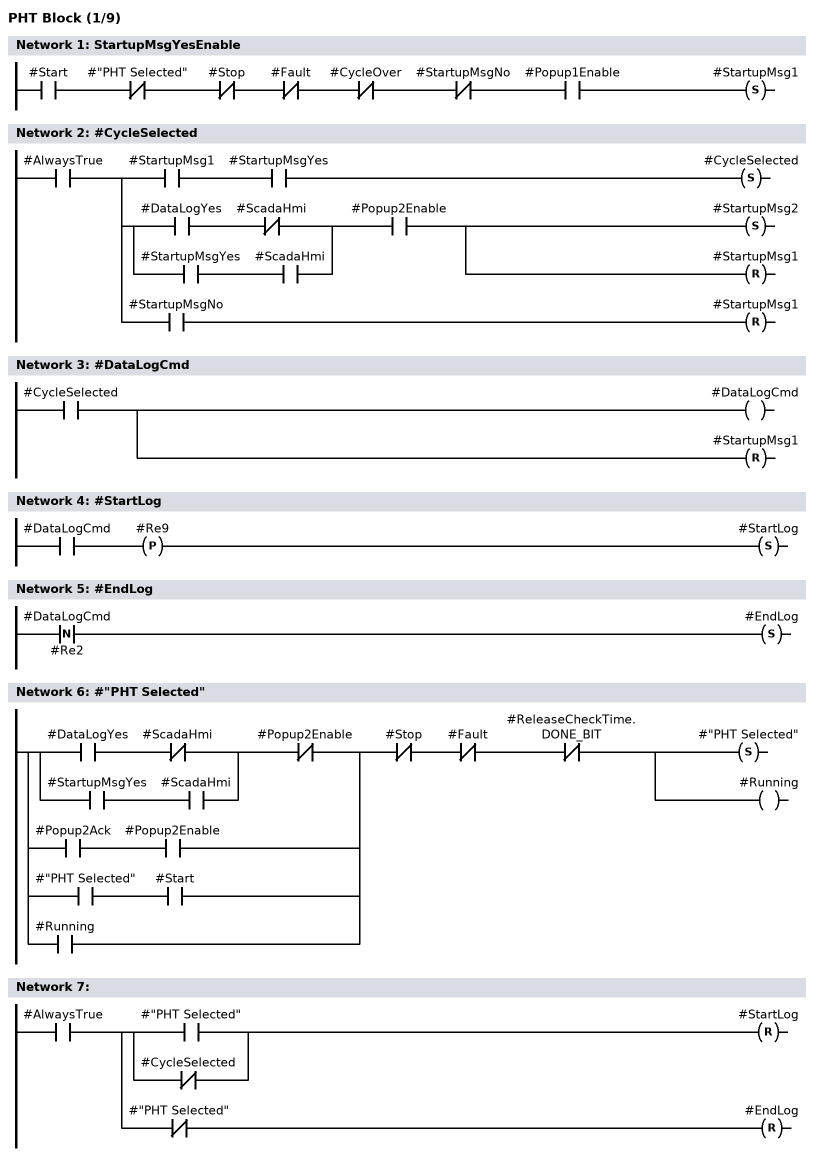
   RUNG wire#powerrail
      Contact( #Start )
      I_Contact( #"PHT Selected" )
      I_Contact( #Stop )
      I_Contact( #Fault )
      I_Contact( #CycleOver )
      I_Contact( #StartupMsgNo )
      Contact( #Popup1Enable )
      S_Coil( #StartupMsg1 )
   END_RUNG
   // the same network as SCL:
   IF #Start AND NOT #"PHT Selected" AND NOT #Stop AND NOT #Fault AND NOT #CycleOver AND NOT #StartupMsgNo AND #Popup1Enable THEN
       #StartupMsg1 := TRUE;
   END_IF;
END_REGION

REGION Network 2: #CycleSelected
   RUNG wire#powerrail
      Contact( #AlwaysTrue )
      wire#w1
      Contact( #StartupMsg1 )
      Contact( #StartupMsgYes )
      S_Coil( #CycleSelected )
   END_RUNG
   RUNG wire#w1
      Contact( #DataLogYes )
      I_Contact( #ScadaHmi )
      wire#w2
      Contact( #Popup2Enable )
      wire#w3
      S_Coil( #StartupMsg2 )
   END_RUNG
   RUNG wire#w1
      Contact( #StartupMsgYes )
      Contact( #ScadaHmi )
   END_RUNG wire#w2
   RUNG wire#w3
      R_Coil( #StartupMsg1 )
   END_RUNG
   RUNG wire#w1
      Contact( #StartupMsgNo )
      R_Coil( #StartupMsg1 )
   END_RUNG
   // the same network as SCL:
   IF #AlwaysTrue AND #StartupMsg1 AND #StartupMsgYes THEN #CycleSelected := TRUE; END_IF;
   IF #AlwaysTrue AND ((#DataLogYes AND NOT #ScadaHmi) OR (#StartupMsgYes AND #ScadaHmi)) AND #Popup2Enable THEN
       #StartupMsg2 := TRUE;
       #StartupMsg1 := FALSE;
   END_IF;
   IF #AlwaysTrue AND #StartupMsgNo THEN #StartupMsg1 := FALSE; END_IF;
END_REGION

REGION Network 3: #DataLogCmd
   RUNG wire#powerrail
      Contact( #CycleSelected )
      wire#w1
      Coil( #DataLogCmd )
   END_RUNG
   RUNG wire#w1
      R_Coil( #StartupMsg1 )
   END_RUNG
   // the same network as SCL:
   #DataLogCmd := #CycleSelected;
   IF #CycleSelected THEN #StartupMsg1 := FALSE; END_IF;
END_REGION

REGION Network 4: #StartLog
   RUNG wire#powerrail
      Contact( #DataLogCmd )
      P_Trig( #Re9 )
      S_Coil( #StartLog )
   END_RUNG
   // the same network as SCL:
   #_w1 := #DataLogCmd AND NOT #Re9;   // rising edge
   #Re9 := #DataLogCmd;
   IF #_w1 THEN #StartLog := TRUE; END_IF;
END_REGION

REGION Network 5: #EndLog
   RUNG wire#powerrail
      N_Contact(operand := #DataLogCmd, bit := #Re2)
      S_Coil( #EndLog )
   END_RUNG
   // the same network as SCL:
   #_w1 := NOT #DataLogCmd AND #Re2;   // falling edge of #DataLogCmd
   #Re2 := #DataLogCmd;
   IF #_w1 THEN #EndLog := TRUE; END_IF;
END_REGION

